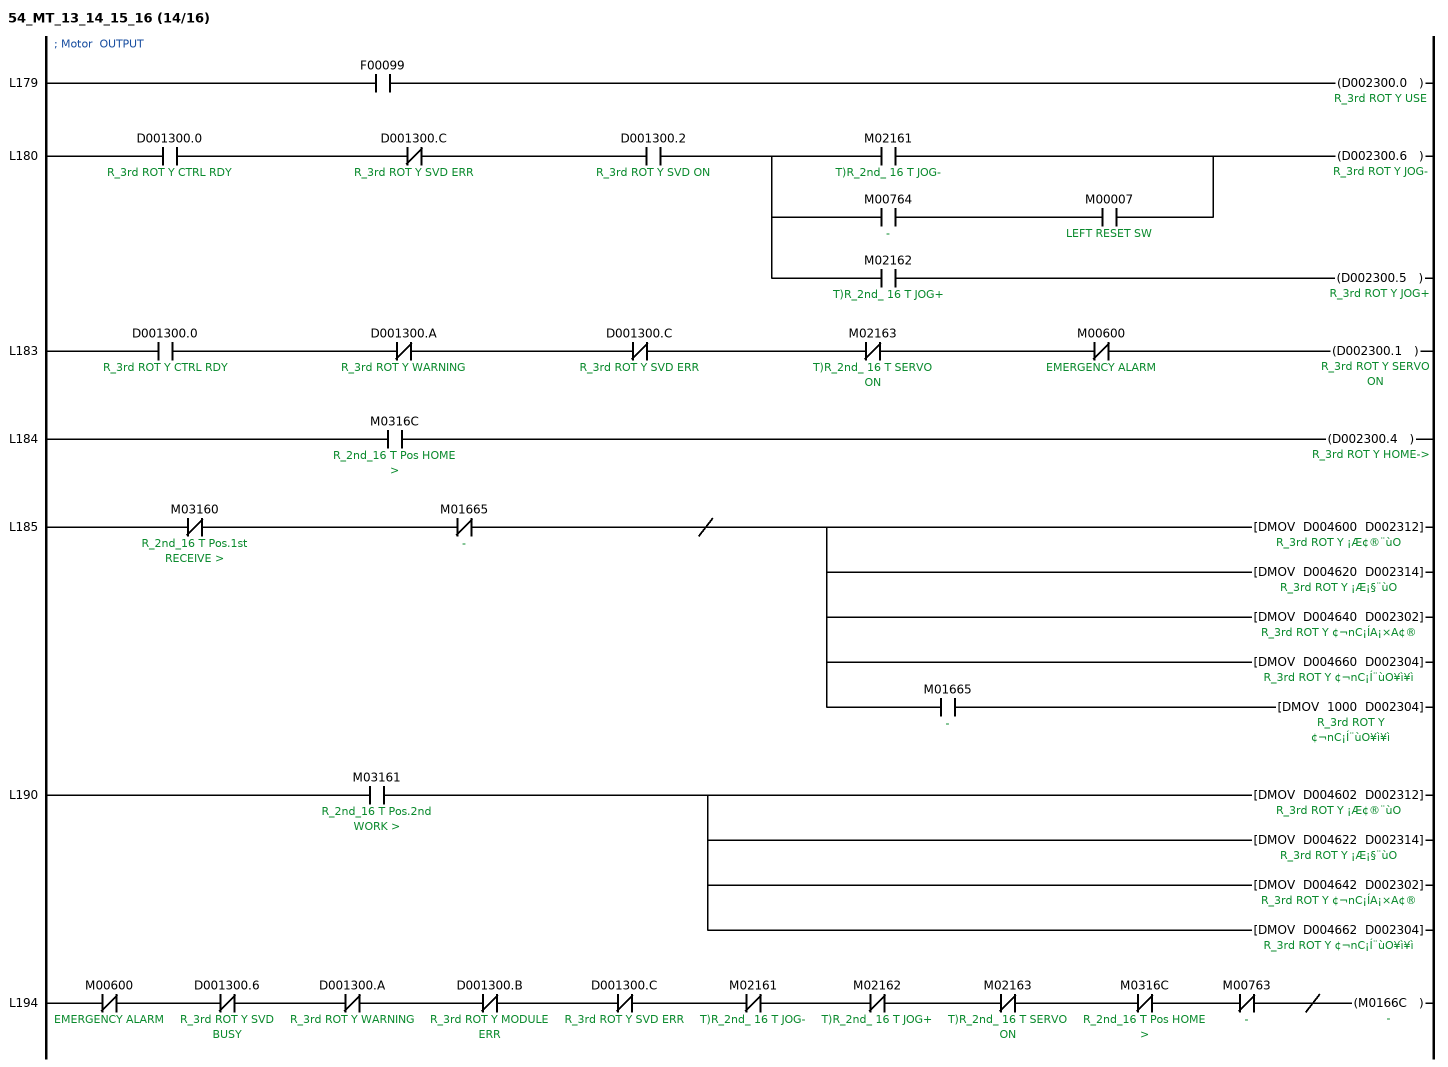
[picture p312: 54_MT_13_14_15_16 rungs L179-L194]
//  Motor  OUTPUT
; L179
LOAD      F00099
OUT       D002300.0	// R_3rd ROT Y USE
; L180
LOAD      D001300.0	// R_3rd ROT Y CTRL RDY
AND NOT   D001300.C	// R_3rd ROT Y SVD ERR
AND       D001300.2	// R_3rd ROT Y SVD ON
MPUSH
LOAD      M02161	// T)R_2nd_ 16 T JOG-
LOAD      M00764	// -
AND       M00007	// LEFT RESET SW
OR LOAD
AND LOAD
OUT       D002300.6	// R_3rd ROT Y JOG-
MPOP
AND       M02162	// T)R_2nd_ 16 T JOG+
OUT       D002300.5	// R_3rd ROT Y JOG+
; L183
LOAD      D001300.0	// R_3rd ROT Y CTRL RDY
AND NOT   D001300.A	// R_3rd ROT Y WARNING
AND NOT   D001300.C	// R_3rd ROT Y SVD ERR
AND NOT   M02163	// T)R_2nd_ 16 T SERVO ON
AND NOT   M00600	// EMERGENCY ALARM
OUT       D002300.1	// R_3rd ROT Y SERVO ON
; L184
LOAD      M0316C	// R_2nd_16 T Pos HOME >
OUT       D002300.4	// R_3rd ROT Y HOME->
; L185
LOAD NOT  M03160	// R_2nd_16 T Pos.1st RECEIVE >
AND NOT   M01665	// -
NOT
DMOV      D004600 D002312	// R_3rd ROT Y ¡Æ¢®¨ùO
DMOV      D004620 D002314	// R_3rd ROT Y ¡Æ¡§¨ùO
DMOV      D004640 D002302	// R_3rd ROT Y ¢¬nC¡ÍA¡×A¢®
DMOV      D004660 D002304	// R_3rd ROT Y ¢¬nC¡Í¨ùO¥ì¥ì
AND       M01665	// -
DMOV      1000 D002304	// R_3rd ROT Y ¢¬nC¡Í¨ùO¥ì¥ì
; L190
LOAD      M03161	// R_2nd_16 T Pos.2nd WORK >
DMOV      D004602 D002312	// R_3rd ROT Y ¡Æ¢®¨ùO
DMOV      D004622 D002314	// R_3rd ROT Y ¡Æ¡§¨ùO
DMOV      D004642 D002302	// R_3rd ROT Y ¢¬nC¡ÍA¡×A¢®
DMOV      D004662 D002304	// R_3rd ROT Y ¢¬nC¡Í¨ùO¥ì¥ì
; L194
LOAD NOT  M00600	// EMERGENCY ALARM
AND NOT   D001300.6	// R_3rd ROT Y SVD BUSY
AND NOT   D001300.A	// R_3rd ROT Y WARNING
AND NOT   D001300.B	// R_3rd ROT Y MODULE ERR
AND NOT   D001300.C	// R_3rd ROT Y SVD ERR
AND NOT   M02161	// T)R_2nd_ 16 T JOG-
AND NOT   M02162	// T)R_2nd_ 16 T JOG+
AND NOT   M02163	// T)R_2nd_ 16 T SERVO ON
AND NOT   M0316C	// R_2nd_16 T Pos HOME >
AND NOT   M00763	// -
NOT
OUT       M0166C	// -

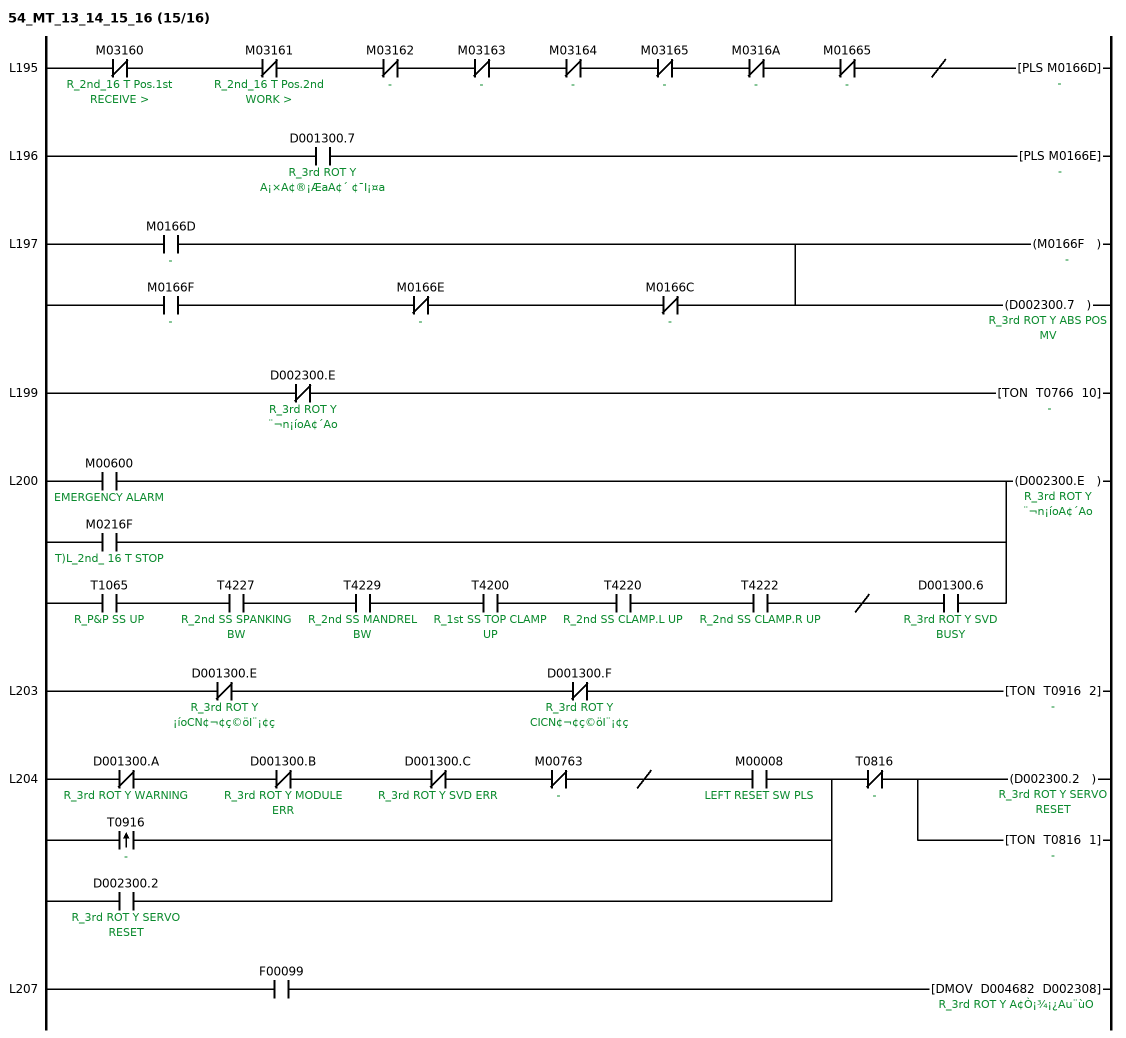
; L195
LOAD NOT  M03160	// R_2nd_16 T Pos.1st RECEIVE >
AND NOT   M03161	// R_2nd_16 T Pos.2nd WORK >
AND NOT   M03162	// -
AND NOT   M03163	// -
AND NOT   M03164	// -
AND NOT   M03165	// -
AND NOT   M0316A	// -
AND NOT   M01665	// -
NOT
OUTP      M0166D	// -
; L196
LOAD      D001300.7	// R_3rd ROT Y A¡×A¢®¡ÆaA¢´ ¢¯I¡¤a
OUTP      M0166E	// -
; L197
LOAD      M0166D	// -
LOAD      M0166F	// -
AND NOT   M0166E	// -
AND NOT   M0166C	// -
OR LOAD
OUT       M0166F	// -
OUT       D002300.7	// R_3rd ROT Y ABS POS MV
; L199
LOAD NOT  D002300.E	// R_3rd ROT Y ¨¬n¡íoA¢´Ao
TON       T0766 10	// -
; L200
LOAD      M00600	// EMERGENCY ALARM
OR        M0216F	// T)L_2nd_ 16 T STOP
LOAD      T1065	// R_P&P SS UP
AND       T4227	// R_2nd SS SPANKING BW
AND       T4229	// R_2nd SS MANDREL BW
AND       T4200	// R_1st SS TOP CLAMP UP
AND       T4220	// R_2nd SS CLAMP.L UP
AND       T4222	// R_2nd SS CLAMP.R UP
NOT
AND       D001300.6	// R_3rd ROT Y SVD BUSY
OR LOAD
OUT       D002300.E	// R_3rd ROT Y ¨¬n¡íoA¢´Ao
; L203
LOAD NOT  D001300.E	// R_3rd ROT Y ¡íoCN¢¬¢ç©öI¨¡¢ç
AND NOT   D001300.F	// R_3rd ROT Y CICN¢¬¢ç©öI¨¡¢ç
TON       T0916 2	// -
; L204
LOAD NOT  D001300.A	// R_3rd ROT Y WARNING
AND NOT   D001300.B	// R_3rd ROT Y MODULE ERR
AND NOT   D001300.C	// R_3rd ROT Y SVD ERR
AND NOT   M00763	// -
NOT
AND       M00008	// LEFT RESET SW PLS
ORP       T0916	// -
OR        D002300.2	// R_3rd ROT Y SERVO RESET
AND NOT   T0816	// -
OUT       D002300.2	// R_3rd ROT Y SERVO RESET
TON       T0816 1	// -
; L207
LOAD      F00099
DMOV      D004682 D002308	// R_3rd ROT Y A¢Ò¡¾¡¿Au¨ùO

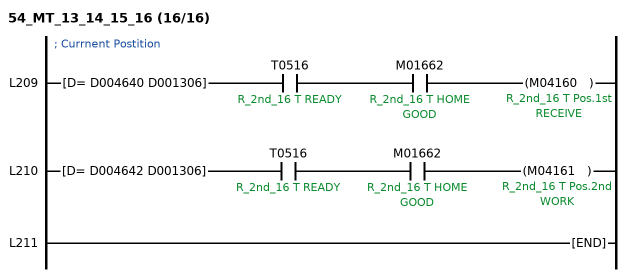
// Currnent Postition
; L209
LOADD=    D004640 D001306
AND       T0516	// R_2nd_16 T READY
AND       M01662	// R_2nd_16 T HOME GOOD
OUT       M04160	// R_2nd_16 T Pos.1st RECEIVE
; L210
LOADD=    D004642 D001306
AND       T0516	// R_2nd_16 T READY
AND       M01662	// R_2nd_16 T HOME GOOD
OUT       M04161	// R_2nd_16 T Pos.2nd WORK
; L211
END

PROGRAM 55_MT_17_18_19_20 (task: ¨ö¨¬A¥ì CA¡¤I¡¾¡¿¡¤¡Í)

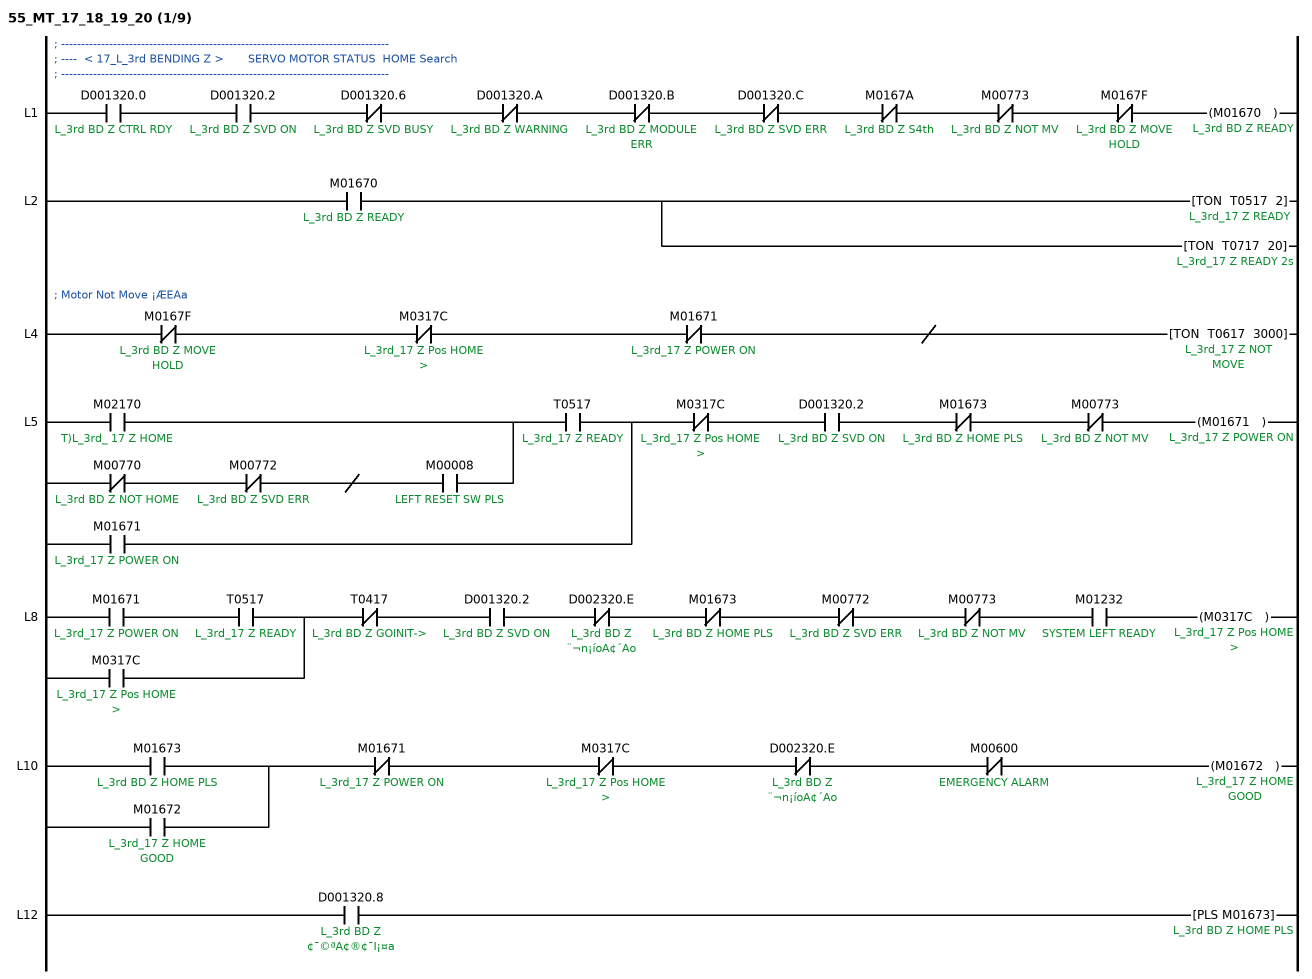
// ----------------------------------------------------------------------------------
// 
// ----  < 17_L_3rd BENDING Z >       SERVO MOTOR STATUS  HOME Search
// 
// ----------------------------------------------------------------------------------
; L1
LOAD      D001320.0	// L_3rd BD Z CTRL RDY
AND       D001320.2	// L_3rd BD Z SVD ON
AND NOT   D001320.6	// L_3rd BD Z SVD BUSY
AND NOT   D001320.A	// L_3rd BD Z WARNING
AND NOT   D001320.B	// L_3rd BD Z MODULE ERR
AND NOT   D001320.C	// L_3rd BD Z SVD ERR
AND NOT   M0167A	// L_3rd BD Z S4th
AND NOT   M00773	// L_3rd BD Z NOT MV
AND NOT   M0167F	// L_3rd BD Z MOVE HOLD
OUT       M01670	// L_3rd BD Z READY
; L2
LOAD      M01670	// L_3rd BD Z READY
TON       T0517 2	// L_3rd_17 Z READY
TON       T0717 20	// L_3rd_17 Z READY 2s
; L4
LOAD NOT  M0167F	// L_3rd BD Z MOVE HOLD
AND NOT   M0317C	// L_3rd_17 Z Pos HOME >
AND NOT   M01671	// L_3rd_17 Z POWER ON
NOT
TON       T0617 3000	// L_3rd_17 Z NOT MOVE
// output comment: Motor Not Move ¡ÆEAa
; L5
LOAD      M02170	// T)L_3rd_ 17 Z HOME
LOAD NOT  M00770	// L_3rd BD Z NOT HOME
AND NOT   M00772	// L_3rd BD Z SVD ERR
NOT
AND       M00008	// LEFT RESET SW PLS
OR LOAD
AND       T0517	// L_3rd_17 Z READY
OR        M01671	// L_3rd_17 Z POWER ON
AND NOT   M0317C	// L_3rd_17 Z Pos HOME >
AND       D001320.2	// L_3rd BD Z SVD ON
AND NOT   M01673	// L_3rd BD Z HOME PLS
AND NOT   M00773	// L_3rd BD Z NOT MV
OUT       M01671	// L_3rd_17 Z POWER ON
; L8
LOAD      M01671	// L_3rd_17 Z POWER ON
AND       T0517	// L_3rd_17 Z READY
OR        M0317C	// L_3rd_17 Z Pos HOME >
AND NOT   T0417	// L_3rd BD Z GOINIT->
AND       D001320.2	// L_3rd BD Z SVD ON
AND NOT   D002320.E	// L_3rd BD Z ¨¬n¡íoA¢´Ao
AND NOT   M01673	// L_3rd BD Z HOME PLS
AND NOT   M00772	// L_3rd BD Z SVD ERR
AND NOT   M00773	// L_3rd BD Z NOT MV
AND       M01232	// SYSTEM LEFT READY
OUT       M0317C	// L_3rd_17 Z Pos HOME >
; L10
LOAD      M01673	// L_3rd BD Z HOME PLS
OR        M01672	// L_3rd_17 Z HOME GOOD
AND NOT   M01671	// L_3rd_17 Z POWER ON
AND NOT   M0317C	// L_3rd_17 Z Pos HOME >
AND NOT   D002320.E	// L_3rd BD Z ¨¬n¡íoA¢´Ao
AND NOT   M00600	// EMERGENCY ALARM
OUT       M01672	// L_3rd_17 Z HOME GOOD
; L12
LOAD      D001320.8	// L_3rd BD Z ¢¯©ªA¢®¢¯I¡¤a
OUTP      M01673	// L_3rd BD Z HOME PLS

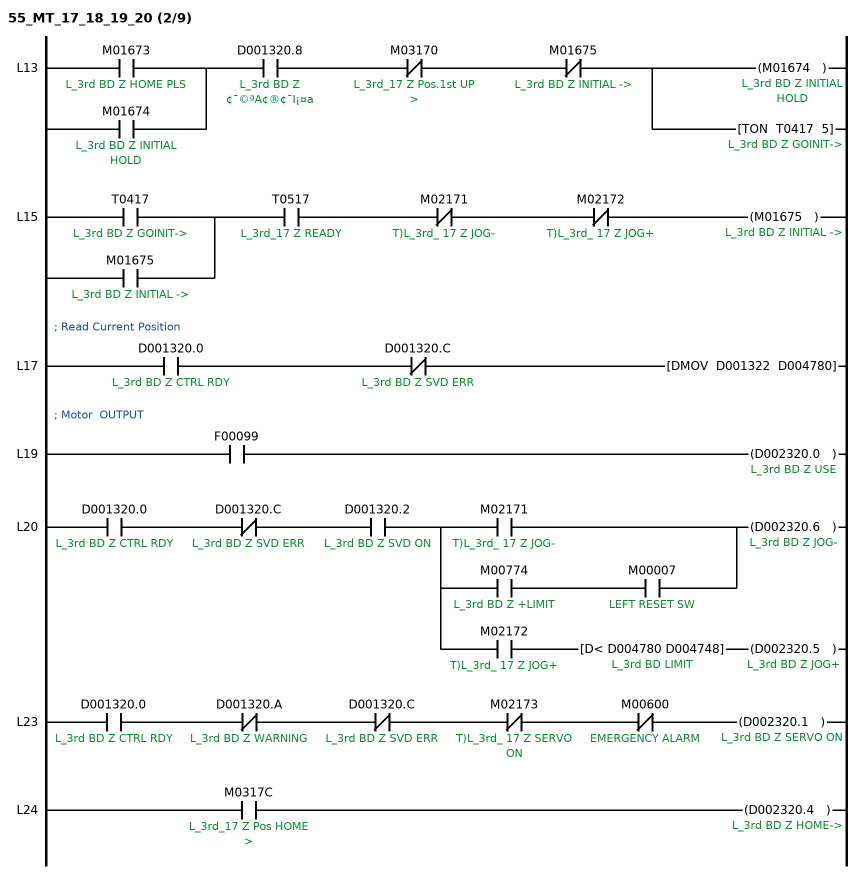
; L13
LOAD      M01673	// L_3rd BD Z HOME PLS
OR        M01674	// L_3rd BD Z INITIAL HOLD
AND       D001320.8	// L_3rd BD Z ¢¯©ªA¢®¢¯I¡¤a
AND NOT   M03170	// L_3rd_17 Z Pos.1st UP >
AND NOT   M01675	// L_3rd BD Z INITIAL ->
OUT       M01674	// L_3rd BD Z INITIAL HOLD
TON       T0417 5	// L_3rd BD Z GOINIT->
; L15
LOAD      T0417	// L_3rd BD Z GOINIT->
OR        M01675	// L_3rd BD Z INITIAL ->
AND       T0517	// L_3rd_17 Z READY
AND NOT   M02171	// T)L_3rd_ 17 Z JOG-
AND NOT   M02172	// T)L_3rd_ 17 Z JOG+
OUT       M01675	// L_3rd BD Z INITIAL ->
; L17
LOAD      D001320.0	// L_3rd BD Z CTRL RDY
AND NOT   D001320.C	// L_3rd BD Z SVD ERR
DMOV      D001322 D004780
// output comment: Read Current Position
//  Motor  OUTPUT
; L19
LOAD      F00099
OUT       D002320.0	// L_3rd BD Z USE
; L20
LOAD      D001320.0	// L_3rd BD Z CTRL RDY
AND NOT   D001320.C	// L_3rd BD Z SVD ERR
AND       D001320.2	// L_3rd BD Z SVD ON
MPUSH
LOAD      M02171	// T)L_3rd_ 17 Z JOG-
LOAD      M00774	// L_3rd BD Z +LIMIT
AND       M00007	// LEFT RESET SW
OR LOAD
AND LOAD
OUT       D002320.6	// L_3rd BD Z JOG-
MPOP
AND       M02172	// T)L_3rd_ 17 Z JOG+
ANDD<     D004780 D004748	// L_3rd BD LIMIT
OUT       D002320.5	// L_3rd BD Z JOG+
; L23
LOAD      D001320.0	// L_3rd BD Z CTRL RDY
AND NOT   D001320.A	// L_3rd BD Z WARNING
AND NOT   D001320.C	// L_3rd BD Z SVD ERR
AND NOT   M02173	// T)L_3rd_ 17 Z SERVO ON
AND NOT   M00600	// EMERGENCY ALARM
OUT       D002320.1	// L_3rd BD Z SERVO ON
; L24
LOAD      M0317C	// L_3rd_17 Z Pos HOME >
OUT       D002320.4	// L_3rd BD Z HOME->

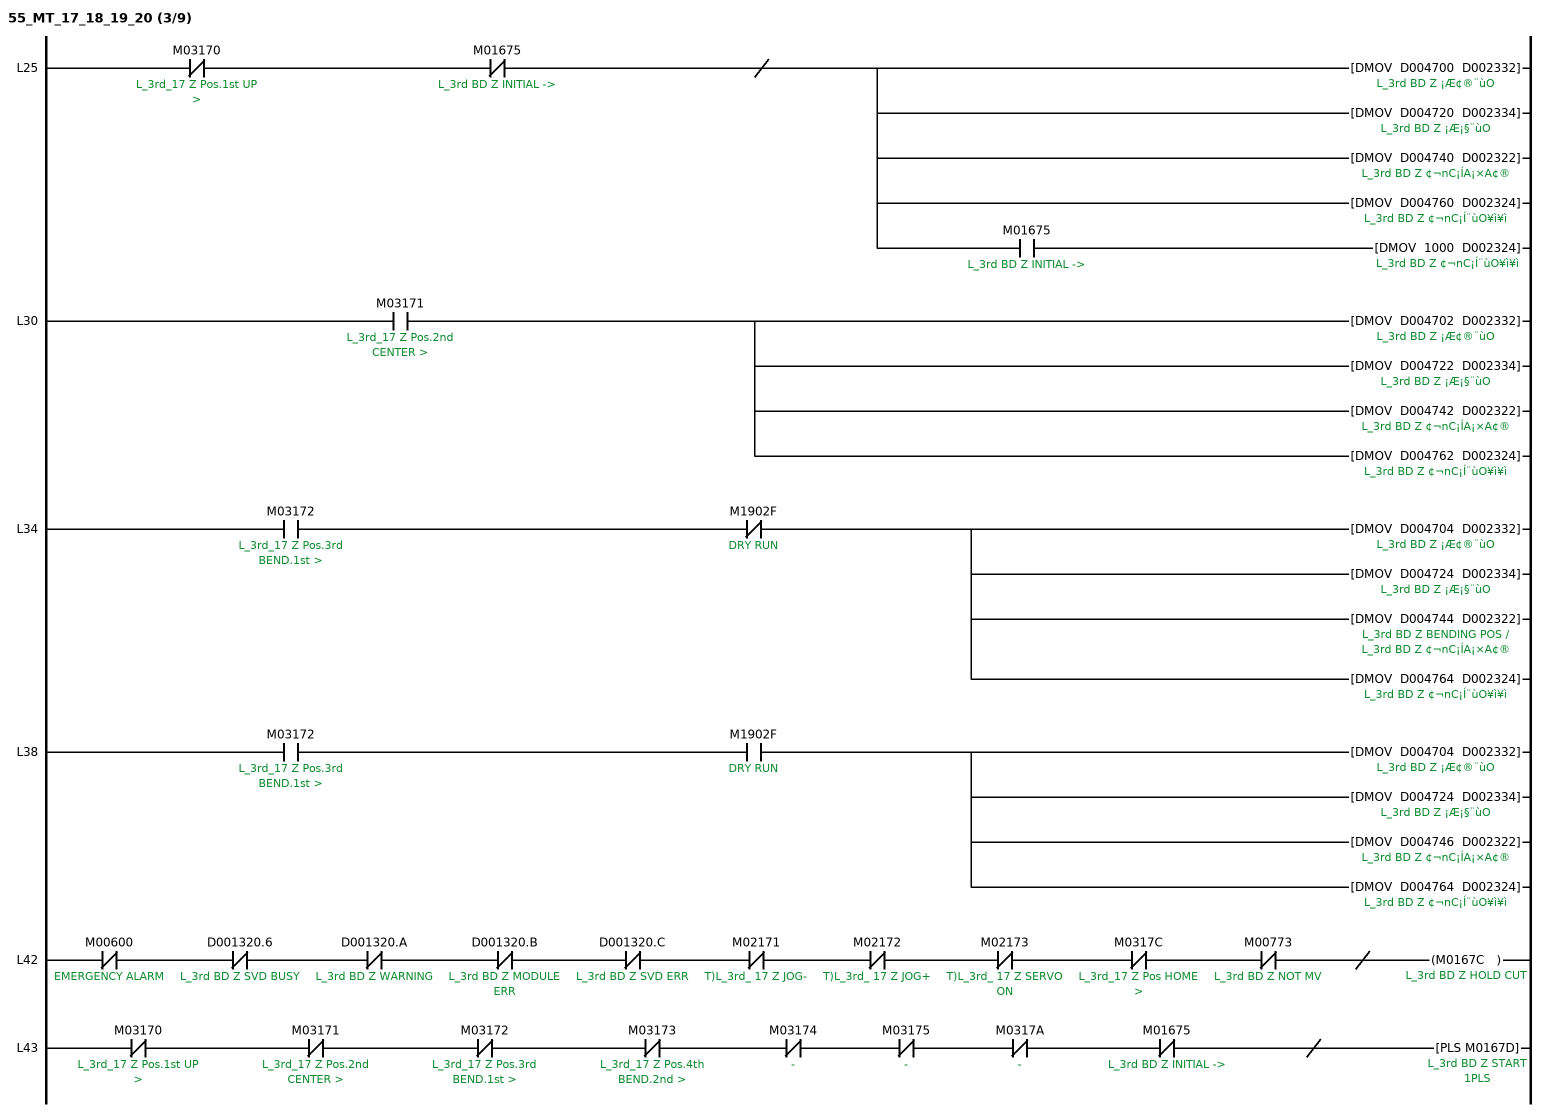
; L25
LOAD NOT  M03170	// L_3rd_17 Z Pos.1st UP >
AND NOT   M01675	// L_3rd BD Z INITIAL ->
NOT
DMOV      D004700 D002332	// L_3rd BD Z ¡Æ¢®¨ùO
DMOV      D004720 D002334	// L_3rd BD Z ¡Æ¡§¨ùO
DMOV      D004740 D002322	// L_3rd BD Z ¢¬nC¡ÍA¡×A¢®
DMOV      D004760 D002324	// L_3rd BD Z ¢¬nC¡Í¨ùO¥ì¥ì
AND       M01675	// L_3rd BD Z INITIAL ->
DMOV      1000 D002324	// L_3rd BD Z ¢¬nC¡Í¨ùO¥ì¥ì
; L30
LOAD      M03171	// L_3rd_17 Z Pos.2nd CENTER >
DMOV      D004702 D002332	// L_3rd BD Z ¡Æ¢®¨ùO
DMOV      D004722 D002334	// L_3rd BD Z ¡Æ¡§¨ùO
DMOV      D004742 D002322	// L_3rd BD Z ¢¬nC¡ÍA¡×A¢®
DMOV      D004762 D002324	// L_3rd BD Z ¢¬nC¡Í¨ùO¥ì¥ì
; L34
LOAD      M03172	// L_3rd_17 Z Pos.3rd BEND.1st >
AND NOT   M1902F	// DRY RUN
DMOV      D004704 D002332	// L_3rd BD Z ¡Æ¢®¨ùO
DMOV      D004724 D002334	// L_3rd BD Z ¡Æ¡§¨ùO
DMOV      D004744 D002322	// L_3rd BD Z BENDING POS / L_3rd BD Z ¢¬nC¡ÍA¡×A¢®
DMOV      D004764 D002324	// L_3rd BD Z ¢¬nC¡Í¨ùO¥ì¥ì
; L38
LOAD      M03172	// L_3rd_17 Z Pos.3rd BEND.1st >
AND       M1902F	// DRY RUN
DMOV      D004704 D002332	// L_3rd BD Z ¡Æ¢®¨ùO
DMOV      D004724 D002334	// L_3rd BD Z ¡Æ¡§¨ùO
DMOV      D004746 D002322	// L_3rd BD Z ¢¬nC¡ÍA¡×A¢®
DMOV      D004764 D002324	// L_3rd BD Z ¢¬nC¡Í¨ùO¥ì¥ì
; L42
LOAD NOT  M00600	// EMERGENCY ALARM
AND NOT   D001320.6	// L_3rd BD Z SVD BUSY
AND NOT   D001320.A	// L_3rd BD Z WARNING
AND NOT   D001320.B	// L_3rd BD Z MODULE ERR
AND NOT   D001320.C	// L_3rd BD Z SVD ERR
AND NOT   M02171	// T)L_3rd_ 17 Z JOG-
AND NOT   M02172	// T)L_3rd_ 17 Z JOG+
AND NOT   M02173	// T)L_3rd_ 17 Z SERVO ON
AND NOT   M0317C	// L_3rd_17 Z Pos HOME >
AND NOT   M00773	// L_3rd BD Z NOT MV
NOT
OUT       M0167C	// L_3rd BD Z HOLD CUT
; L43
LOAD NOT  M03170	// L_3rd_17 Z Pos.1st UP >
AND NOT   M03171	// L_3rd_17 Z Pos.2nd CENTER >
AND NOT   M03172	// L_3rd_17 Z Pos.3rd BEND.1st >
AND NOT   M03173	// L_3rd_17 Z Pos.4th BEND.2nd >
AND NOT   M03174	// -
AND NOT   M03175	// -
AND NOT   M0317A	// -
AND NOT   M01675	// L_3rd BD Z INITIAL ->
NOT
OUTP      M0167D	// L_3rd BD Z START 1PLS

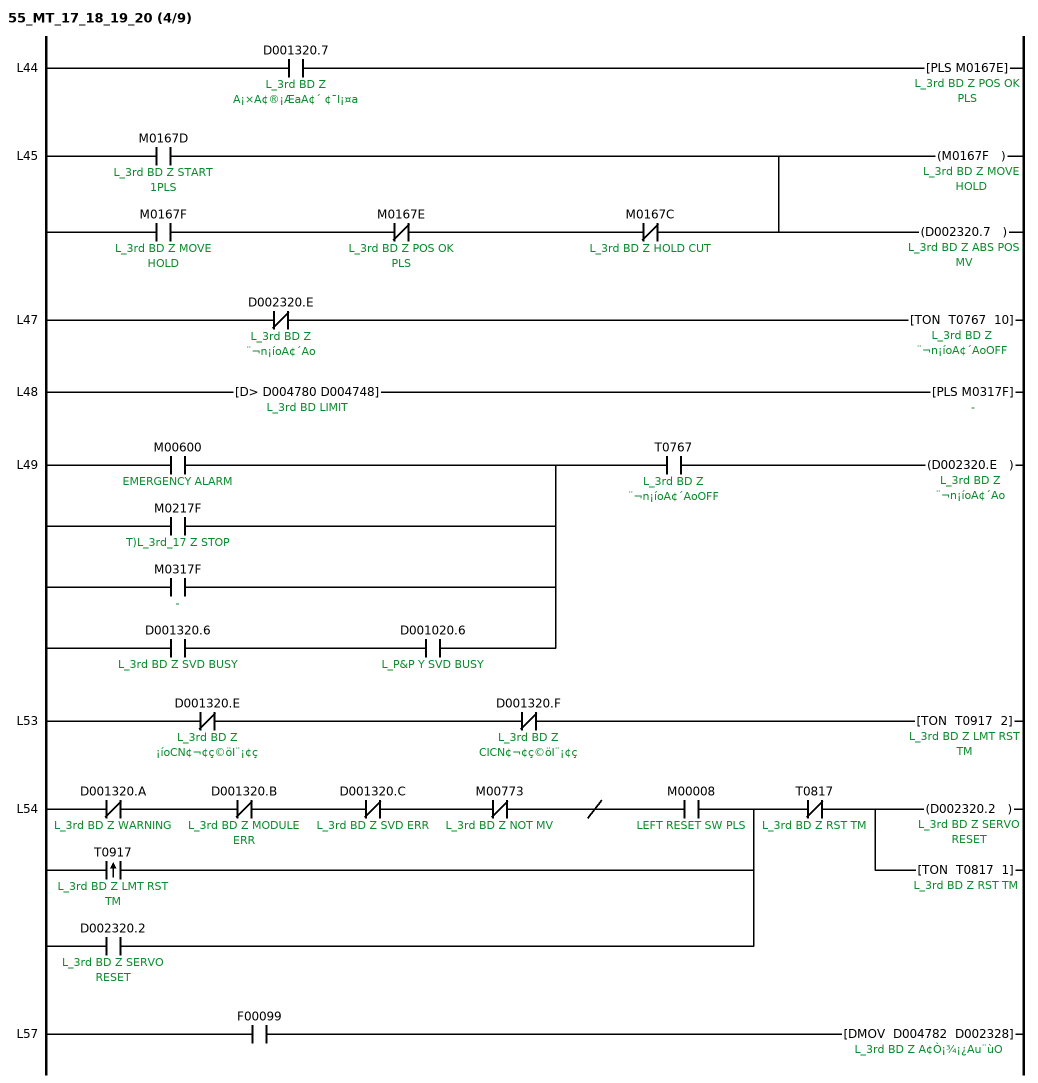
; L44
LOAD      D001320.7	// L_3rd BD Z A¡×A¢®¡ÆaA¢´ ¢¯I¡¤a
OUTP      M0167E	// L_3rd BD Z POS OK PLS
; L45
LOAD      M0167D	// L_3rd BD Z START 1PLS
LOAD      M0167F	// L_3rd BD Z MOVE HOLD
AND NOT   M0167E	// L_3rd BD Z POS OK PLS
AND NOT   M0167C	// L_3rd BD Z HOLD CUT
OR LOAD
OUT       M0167F	// L_3rd BD Z MOVE HOLD
OUT       D002320.7	// L_3rd BD Z ABS POS MV
; L47
LOAD NOT  D002320.E	// L_3rd BD Z ¨¬n¡íoA¢´Ao
TON       T0767 10	// L_3rd BD Z ¨¬n¡íoA¢´AoOFF
; L48
LOADD>    D004780 D004748	// L_3rd BD LIMIT
OUTP      M0317F	// -
; L49
LOAD      M00600	// EMERGENCY ALARM
OR        M0217F	// T)L_3rd_17 Z STOP
OR        M0317F	// -
LOAD      D001320.6	// L_3rd BD Z SVD BUSY
AND       D001020.6	// L_P&P Y SVD BUSY
OR LOAD
AND       T0767	// L_3rd BD Z ¨¬n¡íoA¢´AoOFF
OUT       D002320.E	// L_3rd BD Z ¨¬n¡íoA¢´Ao
; L53
LOAD NOT  D001320.E	// L_3rd BD Z ¡íoCN¢¬¢ç©öI¨¡¢ç
AND NOT   D001320.F	// L_3rd BD Z CICN¢¬¢ç©öI¨¡¢ç
TON       T0917 2	// L_3rd BD Z LMT RST TM
; L54
LOAD NOT  D001320.A	// L_3rd BD Z WARNING
AND NOT   D001320.B	// L_3rd BD Z MODULE ERR
AND NOT   D001320.C	// L_3rd BD Z SVD ERR
AND NOT   M00773	// L_3rd BD Z NOT MV
NOT
AND       M00008	// LEFT RESET SW PLS
ORP       T0917	// L_3rd BD Z LMT RST TM
OR        D002320.2	// L_3rd BD Z SERVO RESET
AND NOT   T0817	// L_3rd BD Z RST TM
OUT       D002320.2	// L_3rd BD Z SERVO RESET
TON       T0817 1	// L_3rd BD Z RST TM
; L57
LOAD      F00099
DMOV      D004782 D002328	// L_3rd BD Z A¢Ò¡¾¡¿Au¨ùO

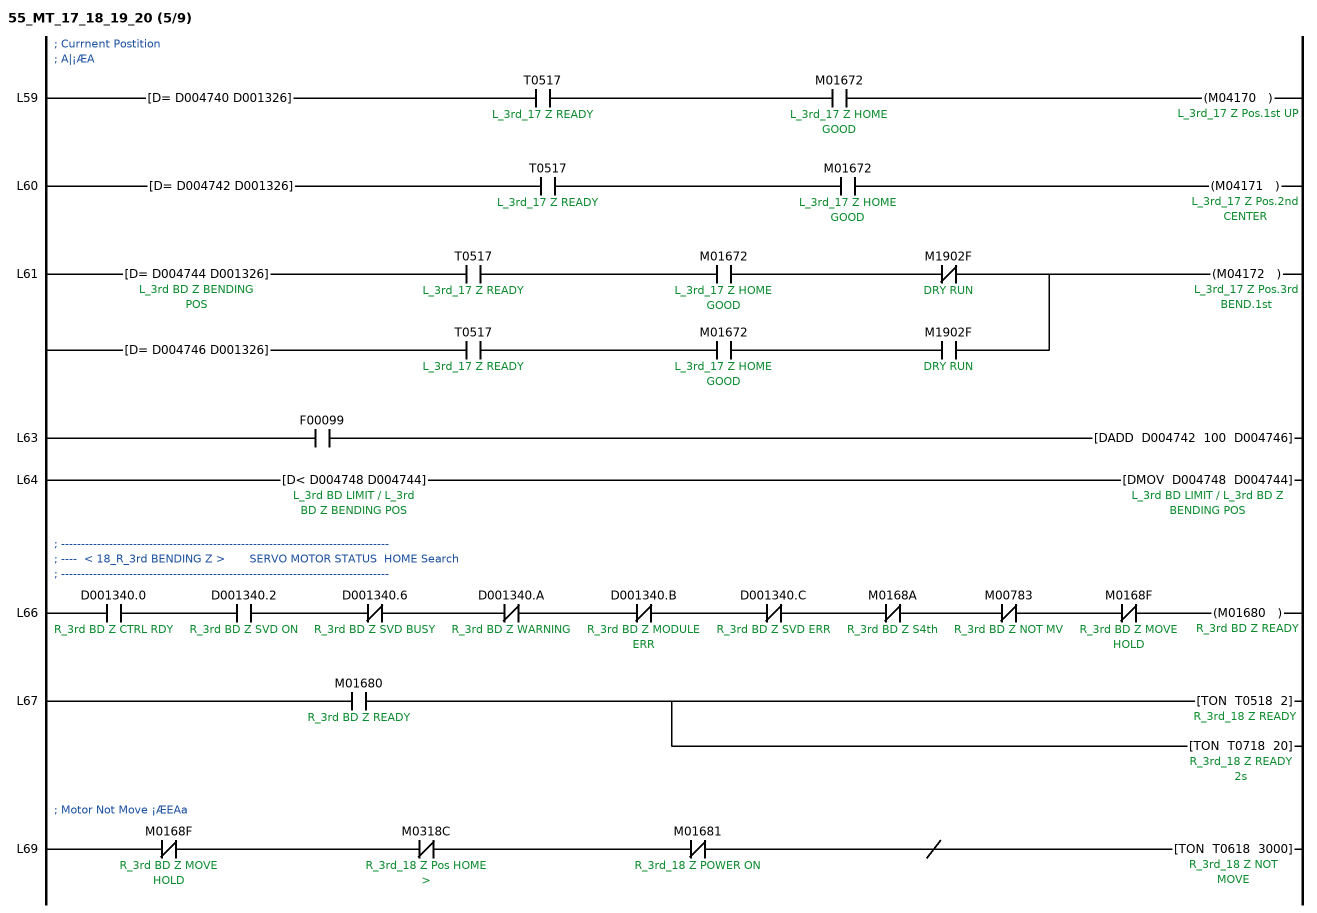
// Currnent Postition
; L59
LOADD=    D004740 D001326
AND       T0517	// L_3rd_17 Z READY
AND       M01672	// L_3rd_17 Z HOME GOOD
OUT       M04170	// L_3rd_17 Z Pos.1st UP
// output comment: A|¡ÆA
; L60
LOADD=    D004742 D001326
AND       T0517	// L_3rd_17 Z READY
AND       M01672	// L_3rd_17 Z HOME GOOD
OUT       M04171	// L_3rd_17 Z Pos.2nd CENTER
; L61
LOADD=    D004744 D001326	// L_3rd BD Z BENDING POS
AND       T0517	// L_3rd_17 Z READY
AND       M01672	// L_3rd_17 Z HOME GOOD
AND NOT   M1902F	// DRY RUN
LOADD=    D004746 D001326
AND       T0517	// L_3rd_17 Z READY
AND       M01672	// L_3rd_17 Z HOME GOOD
AND       M1902F	// DRY RUN
OR LOAD
OUT       M04172	// L_3rd_17 Z Pos.3rd BEND.1st
; L63
LOAD      F00099
DADD      D004742 100 D004746
; L64
LOADD<    D004748 D004744	// L_3rd BD LIMIT / L_3rd BD Z BENDING POS
DMOV      D004748 D004744	// L_3rd BD LIMIT / L_3rd BD Z BENDING POS
// ----------------------------------------------------------------------------------
// 
// ----  < 18_R_3rd BENDING Z >       SERVO MOTOR STATUS  HOME Search
// 
// ----------------------------------------------------------------------------------
; L66
LOAD      D001340.0	// R_3rd BD Z CTRL RDY
AND       D001340.2	// R_3rd BD Z SVD ON
AND NOT   D001340.6	// R_3rd BD Z SVD BUSY
AND NOT   D001340.A	// R_3rd BD Z WARNING
AND NOT   D001340.B	// R_3rd BD Z MODULE ERR
AND NOT   D001340.C	// R_3rd BD Z SVD ERR
AND NOT   M0168A	// R_3rd BD Z S4th
AND NOT   M00783	// R_3rd BD Z NOT MV
AND NOT   M0168F	// R_3rd BD Z MOVE HOLD
OUT       M01680	// R_3rd BD Z READY
; L67
LOAD      M01680	// R_3rd BD Z READY
TON       T0518 2	// R_3rd_18 Z READY
TON       T0718 20	// R_3rd_18 Z READY 2s
; L69
LOAD NOT  M0168F	// R_3rd BD Z MOVE HOLD
AND NOT   M0318C	// R_3rd_18 Z Pos HOME >
AND NOT   M01681	// R_3rd_18 Z POWER ON
NOT
TON       T0618 3000	// R_3rd_18 Z NOT MOVE
// output comment: Motor Not Move ¡ÆEAa

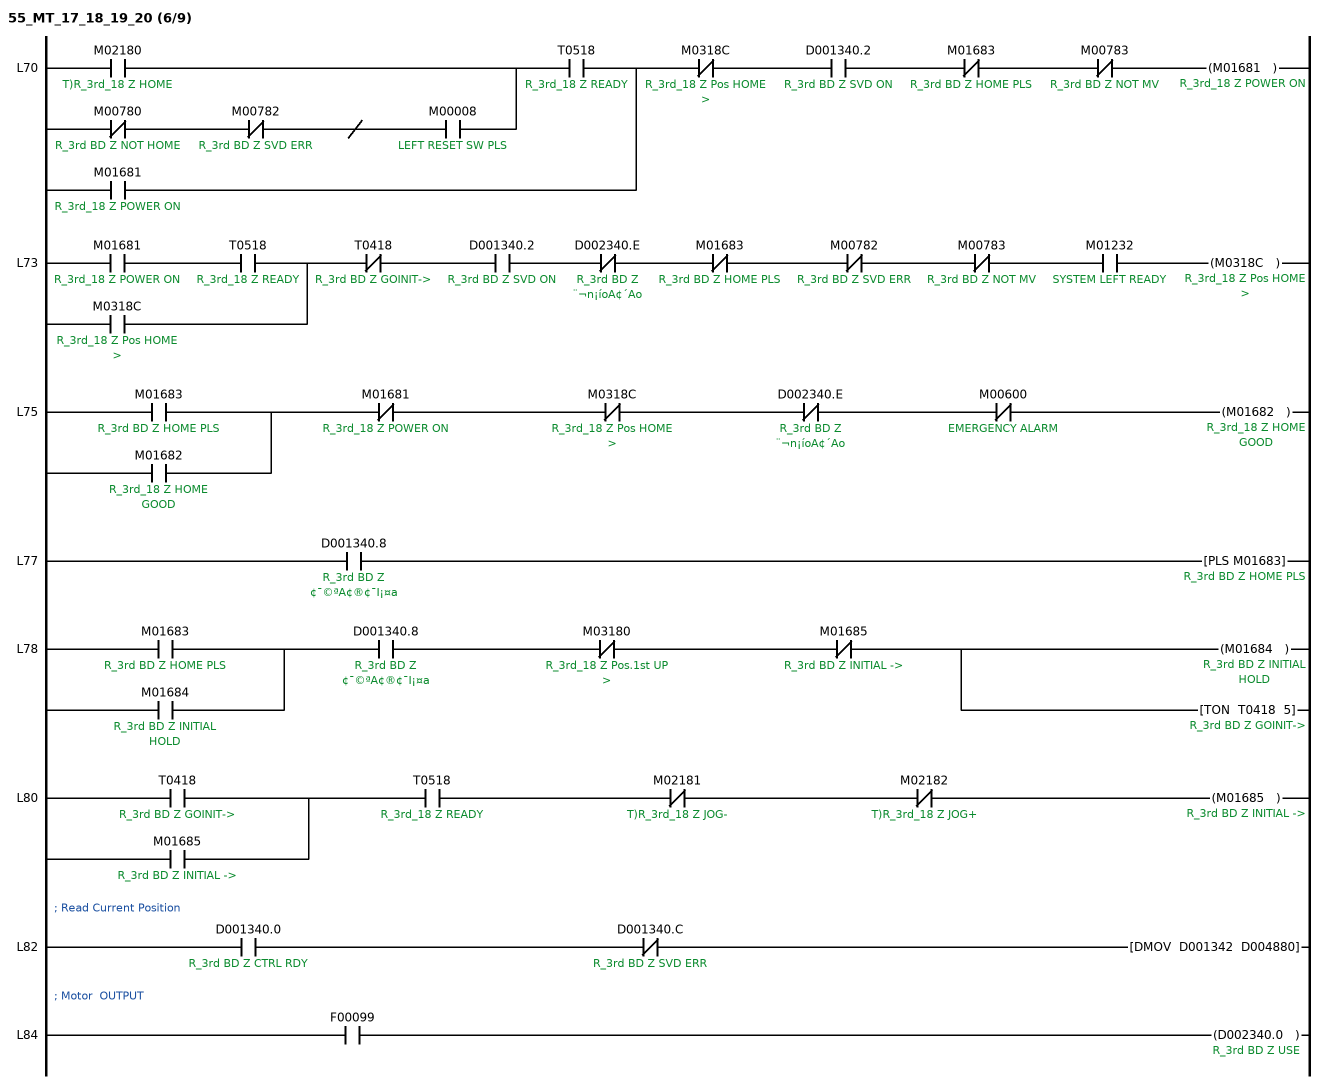
; L70
LOAD      M02180	// T)R_3rd_18 Z HOME
LOAD NOT  M00780	// R_3rd BD Z NOT HOME
AND NOT   M00782	// R_3rd BD Z SVD ERR
NOT
AND       M00008	// LEFT RESET SW PLS
OR LOAD
AND       T0518	// R_3rd_18 Z READY
OR        M01681	// R_3rd_18 Z POWER ON
AND NOT   M0318C	// R_3rd_18 Z Pos HOME >
AND       D001340.2	// R_3rd BD Z SVD ON
AND NOT   M01683	// R_3rd BD Z HOME PLS
AND NOT   M00783	// R_3rd BD Z NOT MV
OUT       M01681	// R_3rd_18 Z POWER ON
; L73
LOAD      M01681	// R_3rd_18 Z POWER ON
AND       T0518	// R_3rd_18 Z READY
OR        M0318C	// R_3rd_18 Z Pos HOME >
AND NOT   T0418	// R_3rd BD Z GOINIT->
AND       D001340.2	// R_3rd BD Z SVD ON
AND NOT   D002340.E	// R_3rd BD Z ¨¬n¡íoA¢´Ao
AND NOT   M01683	// R_3rd BD Z HOME PLS
AND NOT   M00782	// R_3rd BD Z SVD ERR
AND NOT   M00783	// R_3rd BD Z NOT MV
AND       M01232	// SYSTEM LEFT READY
OUT       M0318C	// R_3rd_18 Z Pos HOME >
; L75
LOAD      M01683	// R_3rd BD Z HOME PLS
OR        M01682	// R_3rd_18 Z HOME GOOD
AND NOT   M01681	// R_3rd_18 Z POWER ON
AND NOT   M0318C	// R_3rd_18 Z Pos HOME >
AND NOT   D002340.E	// R_3rd BD Z ¨¬n¡íoA¢´Ao
AND NOT   M00600	// EMERGENCY ALARM
OUT       M01682	// R_3rd_18 Z HOME GOOD
; L77
LOAD      D001340.8	// R_3rd BD Z ¢¯©ªA¢®¢¯I¡¤a
OUTP      M01683	// R_3rd BD Z HOME PLS
; L78
LOAD      M01683	// R_3rd BD Z HOME PLS
OR        M01684	// R_3rd BD Z INITIAL HOLD
AND       D001340.8	// R_3rd BD Z ¢¯©ªA¢®¢¯I¡¤a
AND NOT   M03180	// R_3rd_18 Z Pos.1st UP >
AND NOT   M01685	// R_3rd BD Z INITIAL ->
OUT       M01684	// R_3rd BD Z INITIAL HOLD
TON       T0418 5	// R_3rd BD Z GOINIT->
; L80
LOAD      T0418	// R_3rd BD Z GOINIT->
OR        M01685	// R_3rd BD Z INITIAL ->
AND       T0518	// R_3rd_18 Z READY
AND NOT   M02181	// T)R_3rd_18 Z JOG-
AND NOT   M02182	// T)R_3rd_18 Z JOG+
OUT       M01685	// R_3rd BD Z INITIAL ->
; L82
LOAD      D001340.0	// R_3rd BD Z CTRL RDY
AND NOT   D001340.C	// R_3rd BD Z SVD ERR
DMOV      D001342 D004880
// output comment: Read Current Position
//  Motor  OUTPUT
; L84
LOAD      F00099
OUT       D002340.0	// R_3rd BD Z USE

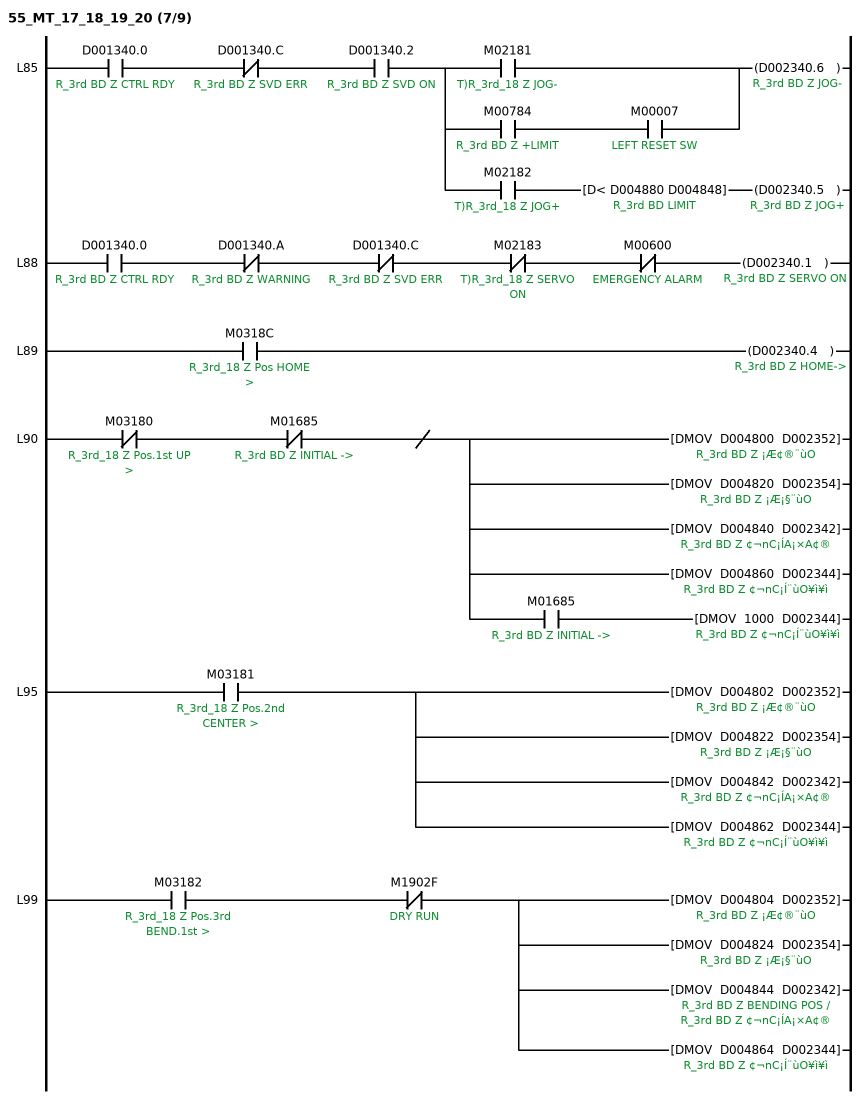
; L85
LOAD      D001340.0	// R_3rd BD Z CTRL RDY
AND NOT   D001340.C	// R_3rd BD Z SVD ERR
AND       D001340.2	// R_3rd BD Z SVD ON
MPUSH
LOAD      M02181	// T)R_3rd_18 Z JOG-
LOAD      M00784	// R_3rd BD Z +LIMIT
AND       M00007	// LEFT RESET SW
OR LOAD
AND LOAD
OUT       D002340.6	// R_3rd BD Z JOG-
MPOP
AND       M02182	// T)R_3rd_18 Z JOG+
ANDD<     D004880 D004848	// R_3rd BD LIMIT
OUT       D002340.5	// R_3rd BD Z JOG+
; L88
LOAD      D001340.0	// R_3rd BD Z CTRL RDY
AND NOT   D001340.A	// R_3rd BD Z WARNING
AND NOT   D001340.C	// R_3rd BD Z SVD ERR
AND NOT   M02183	// T)R_3rd_18 Z SERVO ON
AND NOT   M00600	// EMERGENCY ALARM
OUT       D002340.1	// R_3rd BD Z SERVO ON
; L89
LOAD      M0318C	// R_3rd_18 Z Pos HOME >
OUT       D002340.4	// R_3rd BD Z HOME->
; L90
LOAD NOT  M03180	// R_3rd_18 Z Pos.1st UP >
AND NOT   M01685	// R_3rd BD Z INITIAL ->
NOT
DMOV      D004800 D002352	// R_3rd BD Z ¡Æ¢®¨ùO
DMOV      D004820 D002354	// R_3rd BD Z ¡Æ¡§¨ùO
DMOV      D004840 D002342	// R_3rd BD Z ¢¬nC¡ÍA¡×A¢®
DMOV      D004860 D002344	// R_3rd BD Z ¢¬nC¡Í¨ùO¥ì¥ì
AND       M01685	// R_3rd BD Z INITIAL ->
DMOV      1000 D002344	// R_3rd BD Z ¢¬nC¡Í¨ùO¥ì¥ì
; L95
LOAD      M03181	// R_3rd_18 Z Pos.2nd CENTER >
DMOV      D004802 D002352	// R_3rd BD Z ¡Æ¢®¨ùO
DMOV      D004822 D002354	// R_3rd BD Z ¡Æ¡§¨ùO
DMOV      D004842 D002342	// R_3rd BD Z ¢¬nC¡ÍA¡×A¢®
DMOV      D004862 D002344	// R_3rd BD Z ¢¬nC¡Í¨ùO¥ì¥ì
; L99
LOAD      M03182	// R_3rd_18 Z Pos.3rd BEND.1st >
AND NOT   M1902F	// DRY RUN
DMOV      D004804 D002352	// R_3rd BD Z ¡Æ¢®¨ùO
DMOV      D004824 D002354	// R_3rd BD Z ¡Æ¡§¨ùO
DMOV      D004844 D002342	// R_3rd BD Z BENDING POS / R_3rd BD Z ¢¬nC¡ÍA¡×A¢®
DMOV      D004864 D002344	// R_3rd BD Z ¢¬nC¡Í¨ùO¥ì¥ì

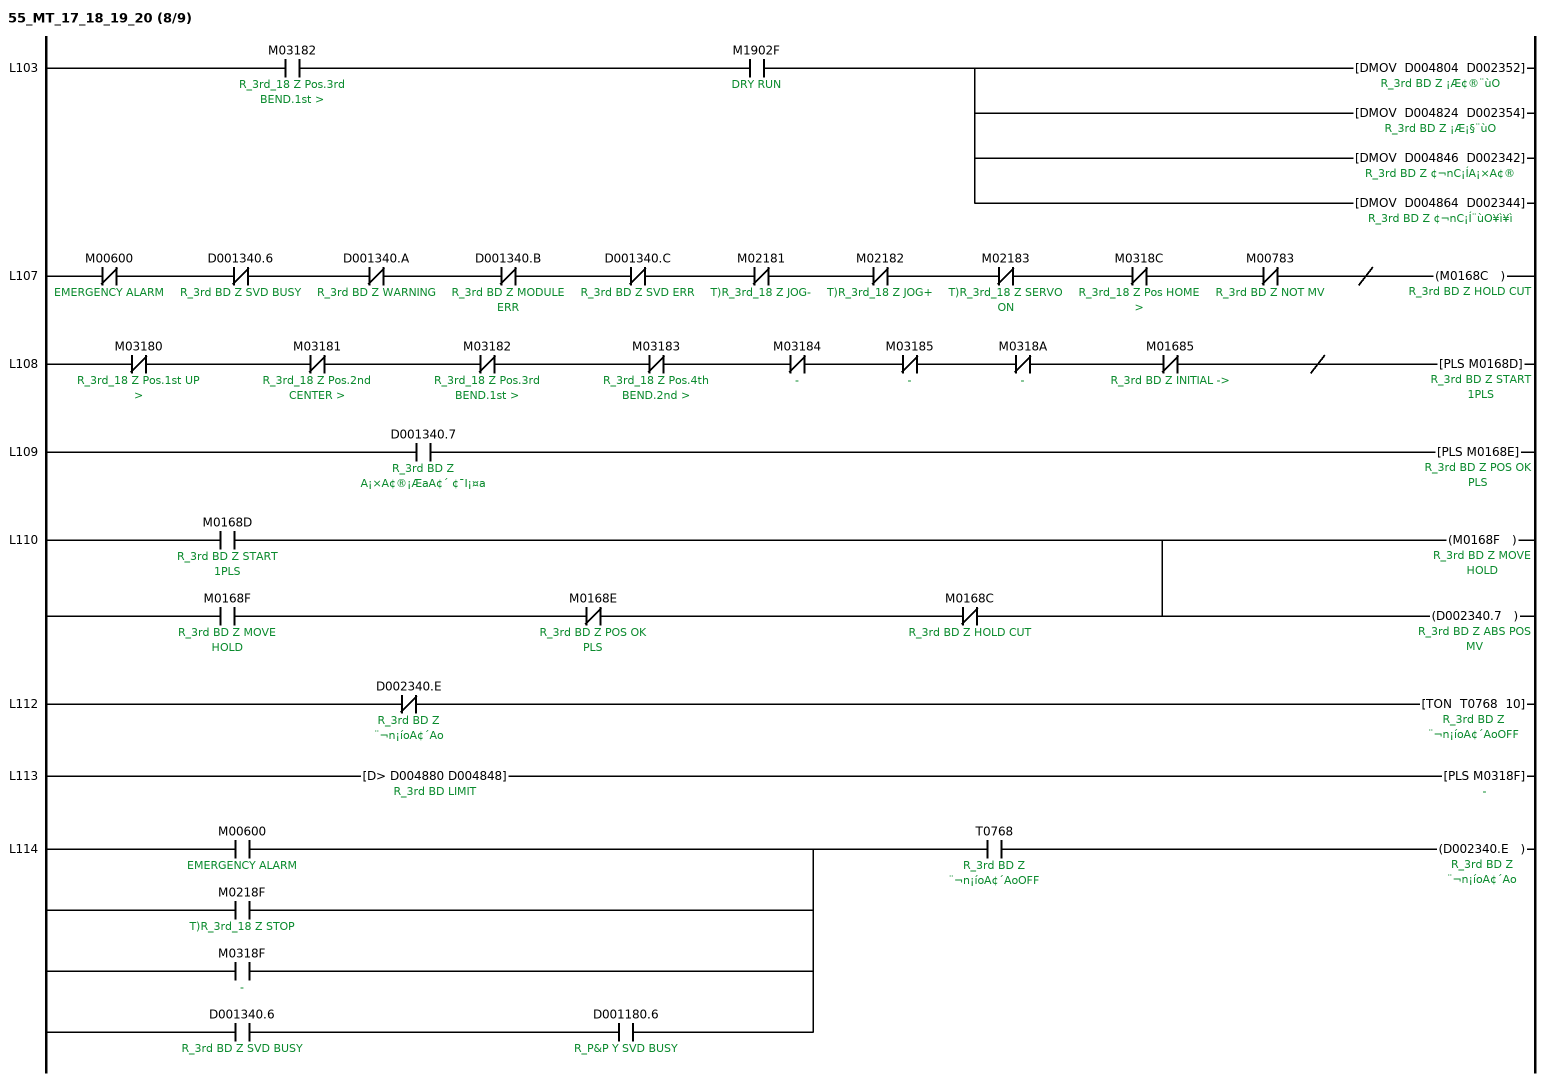
; L103
LOAD      M03182	// R_3rd_18 Z Pos.3rd BEND.1st >
AND       M1902F	// DRY RUN
DMOV      D004804 D002352	// R_3rd BD Z ¡Æ¢®¨ùO
DMOV      D004824 D002354	// R_3rd BD Z ¡Æ¡§¨ùO
DMOV      D004846 D002342	// R_3rd BD Z ¢¬nC¡ÍA¡×A¢®
DMOV      D004864 D002344	// R_3rd BD Z ¢¬nC¡Í¨ùO¥ì¥ì
; L107
LOAD NOT  M00600	// EMERGENCY ALARM
AND NOT   D001340.6	// R_3rd BD Z SVD BUSY
AND NOT   D001340.A	// R_3rd BD Z WARNING
AND NOT   D001340.B	// R_3rd BD Z MODULE ERR
AND NOT   D001340.C	// R_3rd BD Z SVD ERR
AND NOT   M02181	// T)R_3rd_18 Z JOG-
AND NOT   M02182	// T)R_3rd_18 Z JOG+
AND NOT   M02183	// T)R_3rd_18 Z SERVO ON
AND NOT   M0318C	// R_3rd_18 Z Pos HOME >
AND NOT   M00783	// R_3rd BD Z NOT MV
NOT
OUT       M0168C	// R_3rd BD Z HOLD CUT
; L108
LOAD NOT  M03180	// R_3rd_18 Z Pos.1st UP >
AND NOT   M03181	// R_3rd_18 Z Pos.2nd CENTER >
AND NOT   M03182	// R_3rd_18 Z Pos.3rd BEND.1st >
AND NOT   M03183	// R_3rd_18 Z Pos.4th BEND.2nd >
AND NOT   M03184	// -
AND NOT   M03185	// -
AND NOT   M0318A	// -
AND NOT   M01685	// R_3rd BD Z INITIAL ->
NOT
OUTP      M0168D	// R_3rd BD Z START 1PLS
; L109
LOAD      D001340.7	// R_3rd BD Z A¡×A¢®¡ÆaA¢´ ¢¯I¡¤a
OUTP      M0168E	// R_3rd BD Z POS OK PLS
; L110
LOAD      M0168D	// R_3rd BD Z START 1PLS
LOAD      M0168F	// R_3rd BD Z MOVE HOLD
AND NOT   M0168E	// R_3rd BD Z POS OK PLS
AND NOT   M0168C	// R_3rd BD Z HOLD CUT
OR LOAD
OUT       M0168F	// R_3rd BD Z MOVE HOLD
OUT       D002340.7	// R_3rd BD Z ABS POS MV
; L112
LOAD NOT  D002340.E	// R_3rd BD Z ¨¬n¡íoA¢´Ao
TON       T0768 10	// R_3rd BD Z ¨¬n¡íoA¢´AoOFF
; L113
LOADD>    D004880 D004848	// R_3rd BD LIMIT
OUTP      M0318F	// -
; L114
LOAD      M00600	// EMERGENCY ALARM
OR        M0218F	// T)R_3rd_18 Z STOP
OR        M0318F	// -
LOAD      D001340.6	// R_3rd BD Z SVD BUSY
AND       D001180.6	// R_P&P Y SVD BUSY
OR LOAD
AND       T0768	// R_3rd BD Z ¨¬n¡íoA¢´AoOFF
OUT       D002340.E	// R_3rd BD Z ¨¬n¡íoA¢´Ao

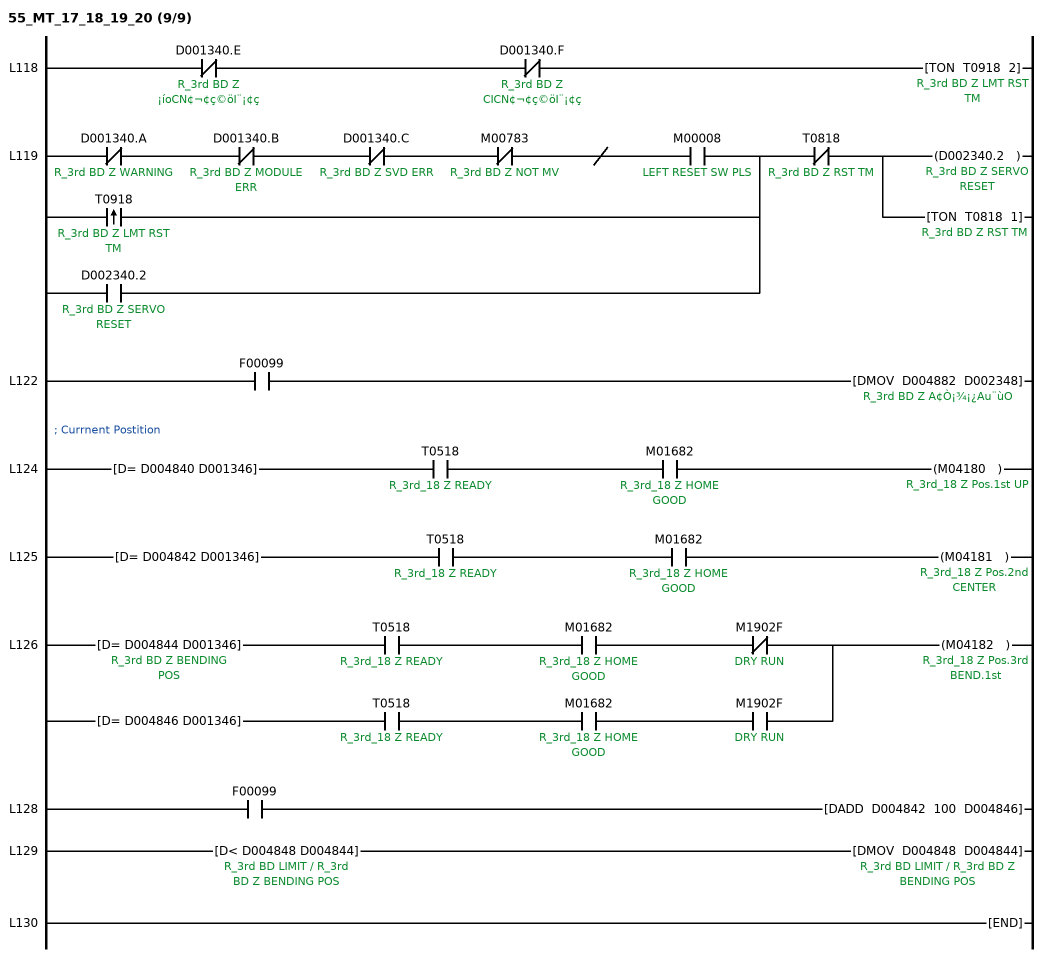
; L118
LOAD NOT  D001340.E	// R_3rd BD Z ¡íoCN¢¬¢ç©öI¨¡¢ç
AND NOT   D001340.F	// R_3rd BD Z CICN¢¬¢ç©öI¨¡¢ç
TON       T0918 2	// R_3rd BD Z LMT RST TM
; L119
LOAD NOT  D001340.A	// R_3rd BD Z WARNING
AND NOT   D001340.B	// R_3rd BD Z MODULE ERR
AND NOT   D001340.C	// R_3rd BD Z SVD ERR
AND NOT   M00783	// R_3rd BD Z NOT MV
NOT
AND       M00008	// LEFT RESET SW PLS
ORP       T0918	// R_3rd BD Z LMT RST TM
OR        D002340.2	// R_3rd BD Z SERVO RESET
AND NOT   T0818	// R_3rd BD Z RST TM
OUT       D002340.2	// R_3rd BD Z SERVO RESET
TON       T0818 1	// R_3rd BD Z RST TM
; L122
LOAD      F00099
DMOV      D004882 D002348	// R_3rd BD Z A¢Ò¡¾¡¿Au¨ùO
// Currnent Postition
; L124
LOADD=    D004840 D001346
AND       T0518	// R_3rd_18 Z READY
AND       M01682	// R_3rd_18 Z HOME GOOD
OUT       M04180	// R_3rd_18 Z Pos.1st UP
; L125
LOADD=    D004842 D001346
AND       T0518	// R_3rd_18 Z READY
AND       M01682	// R_3rd_18 Z HOME GOOD
OUT       M04181	// R_3rd_18 Z Pos.2nd CENTER
; L126
LOADD=    D004844 D001346	// R_3rd BD Z BENDING POS
AND       T0518	// R_3rd_18 Z READY
AND       M01682	// R_3rd_18 Z HOME GOOD
AND NOT   M1902F	// DRY RUN
LOADD=    D004846 D001346
AND       T0518	// R_3rd_18 Z READY
AND       M01682	// R_3rd_18 Z HOME GOOD
AND       M1902F	// DRY RUN
OR LOAD
OUT       M04182	// R_3rd_18 Z Pos.3rd BEND.1st
; L128
LOAD      F00099
DADD      D004842 100 D004846
; L129
LOADD<    D004848 D004844	// R_3rd BD LIMIT / R_3rd BD Z BENDING POS
DMOV      D004848 D004844	// R_3rd BD LIMIT / R_3rd BD Z BENDING POS
; L130
END

PROGRAM 81_OUTPUT (task: ¨ö¨¬A¥ì CA¡¤I¡¾¡¿¡¤¡Í)

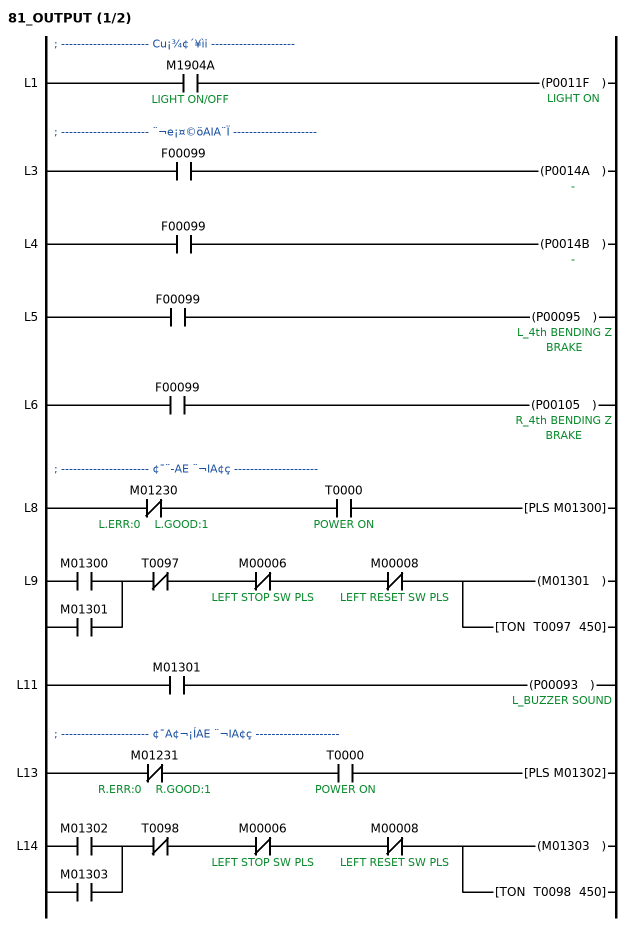
// ---------------------- Cu¡¾¢´¥ìi ---------------------
; L1
LOAD      M1904A	// LIGHT ON/OFF
OUT       P0011F	// LIGHT ON
// ---------------------- ¨¬e¡¤©öAIA¨Ï ---------------------
; L3
LOAD      F00099
OUT       P0014A	// -
; L4
LOAD      F00099
OUT       P0014B	// -
; L5
LOAD      F00099
OUT       P00095	// L_4th BENDING Z BRAKE
; L6
LOAD      F00099
OUT       P00105	// R_4th BENDING Z BRAKE
// ---------------------- ¢¯¨­AE ¨¬IA¢ç ---------------------
; L8
LOAD NOT  M01230	// L.ERR:0    L.GOOD:1
AND       T0000	// POWER ON
OUTP      M01300
; L9
LOAD      M01300
OR        M01301
AND NOT   T0097
AND NOT   M00006	// LEFT STOP SW PLS
AND NOT   M00008	// LEFT RESET SW PLS
OUT       M01301
TON       T0097 450
; L11
LOAD      M01301
OUT       P00093	// L_BUZZER SOUND
// ---------------------- ¢¯A¢¬¡ÍAE ¨¬IA¢ç ---------------------
; L13
LOAD NOT  M01231	// R.ERR:0    R.GOOD:1
AND       T0000	// POWER ON
OUTP      M01302
; L14
LOAD      M01302
OR        M01303
AND NOT   T0098
AND NOT   M00006	// LEFT STOP SW PLS
AND NOT   M00008	// LEFT RESET SW PLS
OUT       M01303
TON       T0098 450

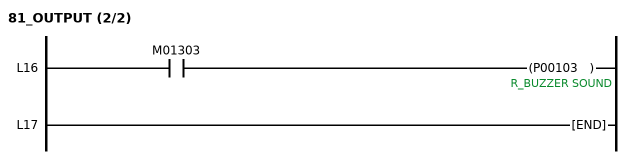
; L16
LOAD      M01303
OUT       P00103	// R_BUZZER SOUND
; L17
END

PROGRAM 82_L_MANUAL (task: ¨ö¨¬A¥ì CA¡¤I¡¾¡¿¡¤¡Í)

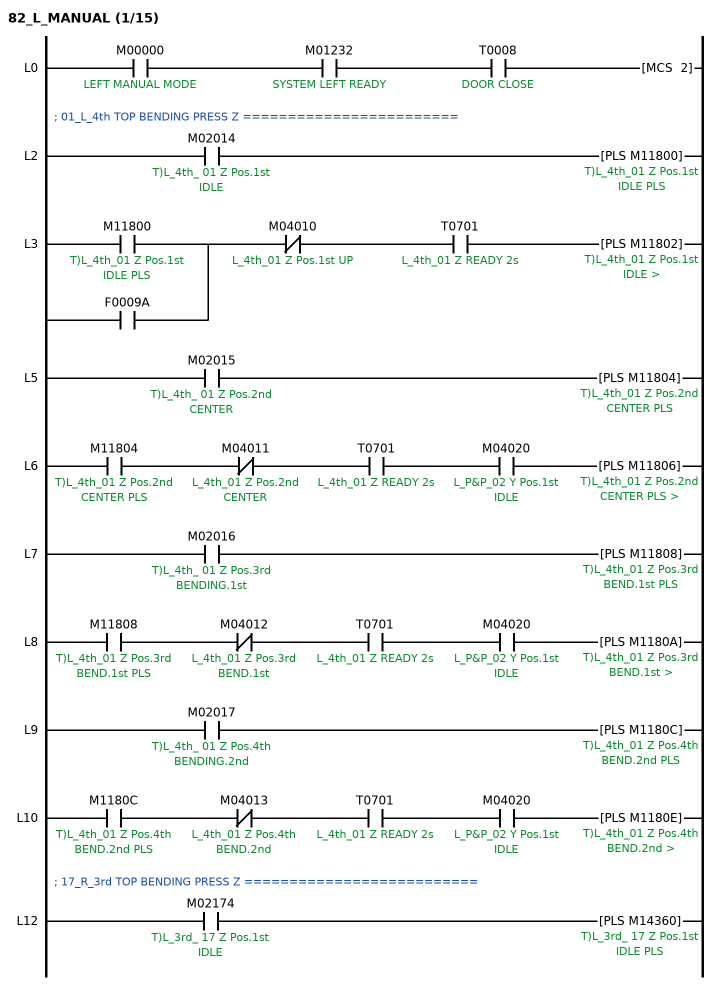
; L0
LOAD      M00000	// LEFT MANUAL MODE
AND       M01232	// SYSTEM LEFT READY
AND       T0008	// DOOR CLOSE
MCS       2
// 01_L_4th TOP BENDING PRESS Z ======================== 
; L2
LOAD      M02014	// T)L_4th_ 01 Z Pos.1st IDLE
OUTP      M11800	// T)L_4th_01 Z Pos.1st IDLE PLS
; L3
LOAD      M11800	// T)L_4th_01 Z Pos.1st IDLE PLS
OR        F0009A
AND NOT   M04010	// L_4th_01 Z Pos.1st UP
AND       T0701	// L_4th_01 Z READY 2s
OUTP      M11802	// T)L_4th_01 Z Pos.1st IDLE >
; L5
LOAD      M02015	// T)L_4th_ 01 Z Pos.2nd CENTER
OUTP      M11804	// T)L_4th_01 Z Pos.2nd CENTER PLS
; L6
LOAD      M11804	// T)L_4th_01 Z Pos.2nd CENTER PLS
AND NOT   M04011	// L_4th_01 Z Pos.2nd CENTER
AND       T0701	// L_4th_01 Z READY 2s
AND       M04020	// L_P&P_02 Y Pos.1st IDLE
OUTP      M11806	// T)L_4th_01 Z Pos.2nd CENTER PLS >
; L7
LOAD      M02016	// T)L_4th_ 01 Z Pos.3rd BENDING.1st
OUTP      M11808	// T)L_4th_01 Z Pos.3rd BEND.1st PLS
; L8
LOAD      M11808	// T)L_4th_01 Z Pos.3rd BEND.1st PLS
AND NOT   M04012	// L_4th_01 Z Pos.3rd BEND.1st
AND       T0701	// L_4th_01 Z READY 2s
AND       M04020	// L_P&P_02 Y Pos.1st IDLE
OUTP      M1180A	// T)L_4th_01 Z Pos.3rd BEND.1st >
; L9
LOAD      M02017	// T)L_4th_ 01 Z Pos.4th BENDING.2nd
OUTP      M1180C	// T)L_4th_01 Z Pos.4th BEND.2nd PLS
; L10
LOAD      M1180C	// T)L_4th_01 Z Pos.4th BEND.2nd PLS
AND NOT   M04013	// L_4th_01 Z Pos.4th BEND.2nd
AND       T0701	// L_4th_01 Z READY 2s
AND       M04020	// L_P&P_02 Y Pos.1st IDLE
OUTP      M1180E	// T)L_4th_01 Z Pos.4th BEND.2nd >
// 17_R_3rd TOP BENDING PRESS Z ==========================
; L12
LOAD      M02174	// T)L_3rd_ 17 Z Pos.1st IDLE
OUTP      M14360	// T)L_3rd_ 17 Z Pos.1st IDLE PLS

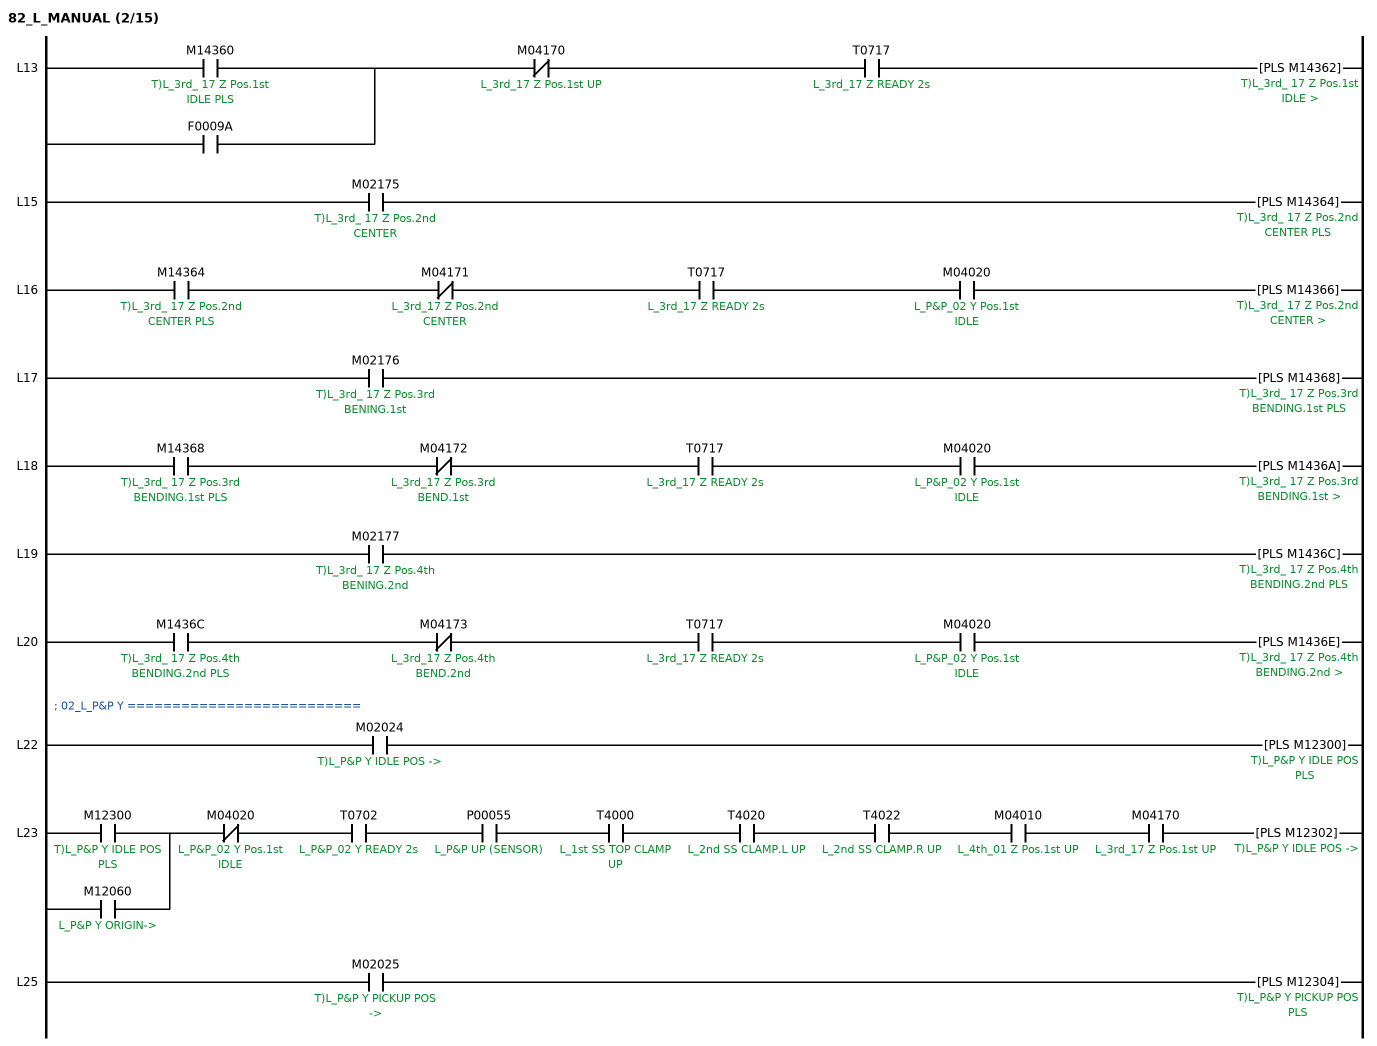
; L13
LOAD      M14360	// T)L_3rd_ 17 Z Pos.1st IDLE PLS
OR        F0009A
AND NOT   M04170	// L_3rd_17 Z Pos.1st UP
AND       T0717	// L_3rd_17 Z READY 2s
OUTP      M14362	// T)L_3rd_ 17 Z Pos.1st IDLE >
; L15
LOAD      M02175	// T)L_3rd_ 17 Z Pos.2nd CENTER
OUTP      M14364	// T)L_3rd_ 17 Z Pos.2nd CENTER PLS
; L16
LOAD      M14364	// T)L_3rd_ 17 Z Pos.2nd CENTER PLS
AND NOT   M04171	// L_3rd_17 Z Pos.2nd CENTER
AND       T0717	// L_3rd_17 Z READY 2s
AND       M04020	// L_P&P_02 Y Pos.1st IDLE
OUTP      M14366	// T)L_3rd_ 17 Z Pos.2nd CENTER >
; L17
LOAD      M02176	// T)L_3rd_ 17 Z Pos.3rd BENING.1st
OUTP      M14368	// T)L_3rd_ 17 Z Pos.3rd BENDING.1st PLS
; L18
LOAD      M14368	// T)L_3rd_ 17 Z Pos.3rd BENDING.1st PLS
AND NOT   M04172	// L_3rd_17 Z Pos.3rd BEND.1st
AND       T0717	// L_3rd_17 Z READY 2s
AND       M04020	// L_P&P_02 Y Pos.1st IDLE
OUTP      M1436A	// T)L_3rd_ 17 Z Pos.3rd BENDING.1st >
; L19
LOAD      M02177	// T)L_3rd_ 17 Z Pos.4th BENING.2nd
OUTP      M1436C	// T)L_3rd_ 17 Z Pos.4th BENDING.2nd PLS
; L20
LOAD      M1436C	// T)L_3rd_ 17 Z Pos.4th BENDING.2nd PLS
AND NOT   M04173	// L_3rd_17 Z Pos.4th BEND.2nd
AND       T0717	// L_3rd_17 Z READY 2s
AND       M04020	// L_P&P_02 Y Pos.1st IDLE
OUTP      M1436E	// T)L_3rd_ 17 Z Pos.4th BENDING.2nd >
// 02_L_P&P Y ==========================
; L22
LOAD      M02024	// T)L_P&P Y IDLE POS ->
OUTP      M12300	// T)L_P&P Y IDLE POS PLS
; L23
LOAD      M12300	// T)L_P&P Y IDLE POS PLS
OR        M12060	// L_P&P Y ORIGIN->
AND NOT   M04020	// L_P&P_02 Y Pos.1st IDLE
AND       T0702	// L_P&P_02 Y READY 2s
AND       P00055	// L_P&P UP (SENSOR)
AND       T4000	// L_1st SS TOP CLAMP    UP
AND       T4020	// L_2nd SS CLAMP.L UP
AND       T4022	// L_2nd SS CLAMP.R UP
AND       M04010	// L_4th_01 Z Pos.1st UP
AND       M04170	// L_3rd_17 Z Pos.1st UP
OUTP      M12302	// T)L_P&P Y IDLE POS ->
; L25
LOAD      M02025	// T)L_P&P Y PICKUP POS ->
OUTP      M12304	// T)L_P&P Y PICKUP POS PLS

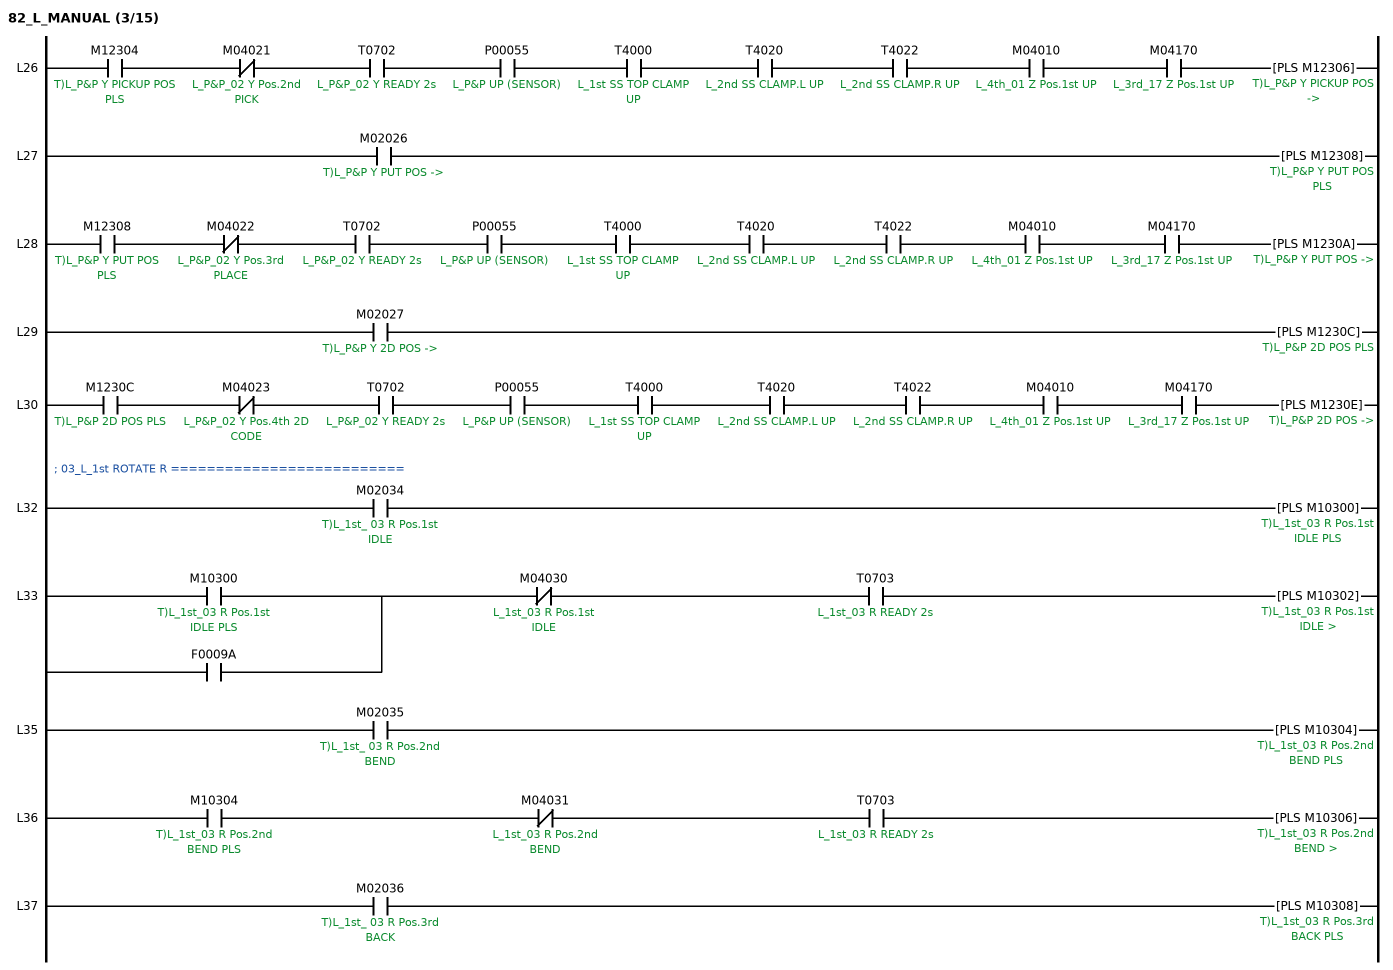
; L26
LOAD      M12304	// T)L_P&P Y PICKUP POS PLS
AND NOT   M04021	// L_P&P_02 Y Pos.2nd PICK
AND       T0702	// L_P&P_02 Y READY 2s
AND       P00055	// L_P&P UP (SENSOR)
AND       T4000	// L_1st SS TOP CLAMP    UP
AND       T4020	// L_2nd SS CLAMP.L UP
AND       T4022	// L_2nd SS CLAMP.R UP
AND       M04010	// L_4th_01 Z Pos.1st UP
AND       M04170	// L_3rd_17 Z Pos.1st UP
OUTP      M12306	// T)L_P&P Y PICKUP POS ->
; L27
LOAD      M02026	// T)L_P&P Y PUT POS ->
OUTP      M12308	// T)L_P&P Y PUT POS PLS
; L28
LOAD      M12308	// T)L_P&P Y PUT POS PLS
AND NOT   M04022	// L_P&P_02 Y Pos.3rd PLACE
AND       T0702	// L_P&P_02 Y READY 2s
AND       P00055	// L_P&P UP (SENSOR)
AND       T4000	// L_1st SS TOP CLAMP    UP
AND       T4020	// L_2nd SS CLAMP.L UP
AND       T4022	// L_2nd SS CLAMP.R UP
AND       M04010	// L_4th_01 Z Pos.1st UP
AND       M04170	// L_3rd_17 Z Pos.1st UP
OUTP      M1230A	// T)L_P&P Y PUT POS ->
; L29
LOAD      M02027	// T)L_P&P Y 2D POS ->
OUTP      M1230C	// T)L_P&P 2D POS PLS
; L30
LOAD      M1230C	// T)L_P&P 2D POS PLS
AND NOT   M04023	// L_P&P_02 Y Pos.4th 2D CODE
AND       T0702	// L_P&P_02 Y READY 2s
AND       P00055	// L_P&P UP (SENSOR)
AND       T4000	// L_1st SS TOP CLAMP    UP
AND       T4020	// L_2nd SS CLAMP.L UP
AND       T4022	// L_2nd SS CLAMP.R UP
AND       M04010	// L_4th_01 Z Pos.1st UP
AND       M04170	// L_3rd_17 Z Pos.1st UP
OUTP      M1230E	// T)L_P&P 2D POS ->
// 03_L_1st ROTATE R ==========================
; L32
LOAD      M02034	// T)L_1st_ 03 R Pos.1st IDLE
OUTP      M10300	// T)L_1st_03 R Pos.1st IDLE PLS
; L33
LOAD      M10300	// T)L_1st_03 R Pos.1st IDLE PLS
OR        F0009A
AND NOT   M04030	// L_1st_03 R Pos.1st IDLE
AND       T0703	// L_1st_03 R READY 2s
OUTP      M10302	// T)L_1st_03 R Pos.1st IDLE >
; L35
LOAD      M02035	// T)L_1st_ 03 R Pos.2nd BEND
OUTP      M10304	// T)L_1st_03 R Pos.2nd BEND PLS
; L36
LOAD      M10304	// T)L_1st_03 R Pos.2nd BEND PLS
AND NOT   M04031	// L_1st_03 R Pos.2nd BEND
AND       T0703	// L_1st_03 R READY 2s
OUTP      M10306	// T)L_1st_03 R Pos.2nd BEND >
; L37
LOAD      M02036	// T)L_1st_ 03 R Pos.3rd BACK
OUTP      M10308	// T)L_1st_03 R Pos.3rd BACK PLS

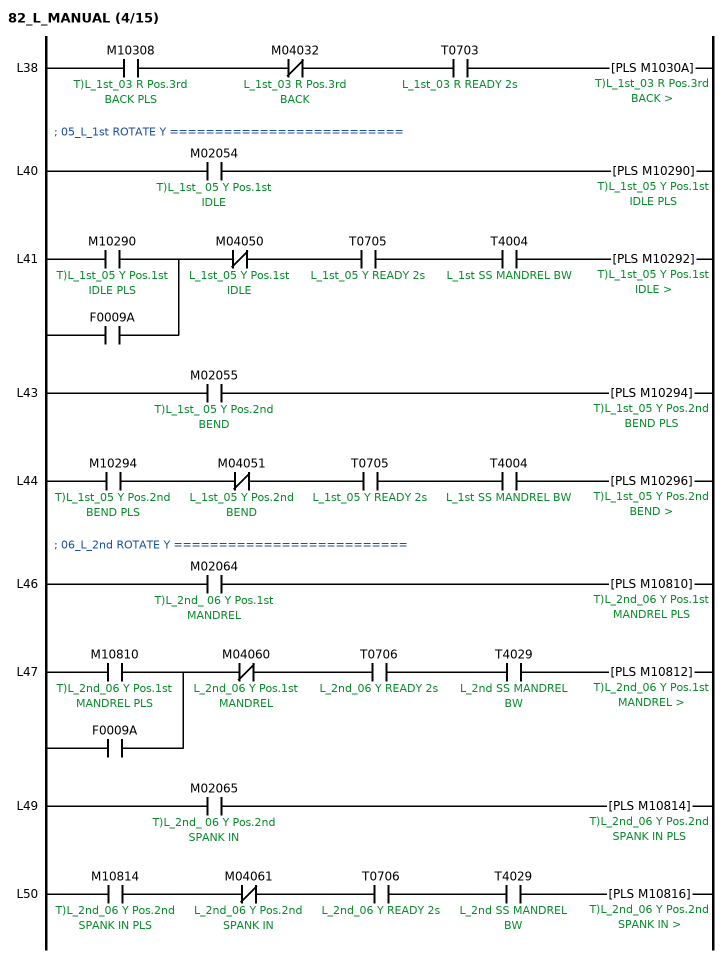
; L38
LOAD      M10308	// T)L_1st_03 R Pos.3rd BACK PLS
AND NOT   M04032	// L_1st_03 R Pos.3rd BACK
AND       T0703	// L_1st_03 R READY 2s
OUTP      M1030A	// T)L_1st_03 R Pos.3rd BACK >
// 05_L_1st ROTATE Y ==========================
; L40
LOAD      M02054	// T)L_1st_ 05 Y Pos.1st IDLE
OUTP      M10290	// T)L_1st_05 Y Pos.1st IDLE PLS
; L41
LOAD      M10290	// T)L_1st_05 Y Pos.1st IDLE PLS
OR        F0009A
AND NOT   M04050	// L_1st_05 Y Pos.1st IDLE
AND       T0705	// L_1st_05 Y READY 2s
AND       T4004	// L_1st SS MANDREL BW
OUTP      M10292	// T)L_1st_05 Y Pos.1st IDLE >
; L43
LOAD      M02055	// T)L_1st_ 05 Y Pos.2nd BEND
OUTP      M10294	// T)L_1st_05 Y Pos.2nd BEND PLS
; L44
LOAD      M10294	// T)L_1st_05 Y Pos.2nd BEND PLS
AND NOT   M04051	// L_1st_05 Y Pos.2nd BEND
AND       T0705	// L_1st_05 Y READY 2s
AND       T4004	// L_1st SS MANDREL BW
OUTP      M10296	// T)L_1st_05 Y Pos.2nd BEND >
// 06_L_2nd ROTATE Y ==========================
; L46
LOAD      M02064	// T)L_2nd_ 06 Y Pos.1st MANDREL
OUTP      M10810	// T)L_2nd_06 Y Pos.1st MANDREL PLS
; L47
LOAD      M10810	// T)L_2nd_06 Y Pos.1st MANDREL PLS
OR        F0009A
AND NOT   M04060	// L_2nd_06 Y Pos.1st MANDREL
AND       T0706	// L_2nd_06 Y READY 2s
AND       T4029	// L_2nd SS MANDREL BW
OUTP      M10812	// T)L_2nd_06 Y Pos.1st MANDREL >
; L49
LOAD      M02065	// T)L_2nd_ 06 Y Pos.2nd SPANK IN
OUTP      M10814	// T)L_2nd_06 Y Pos.2nd SPANK IN PLS
; L50
LOAD      M10814	// T)L_2nd_06 Y Pos.2nd SPANK IN PLS
AND NOT   M04061	// L_2nd_06 Y Pos.2nd SPANK IN
AND       T0706	// L_2nd_06 Y READY 2s
AND       T4029	// L_2nd SS MANDREL BW
OUTP      M10816	// T)L_2nd_06 Y Pos.2nd SPANK IN >

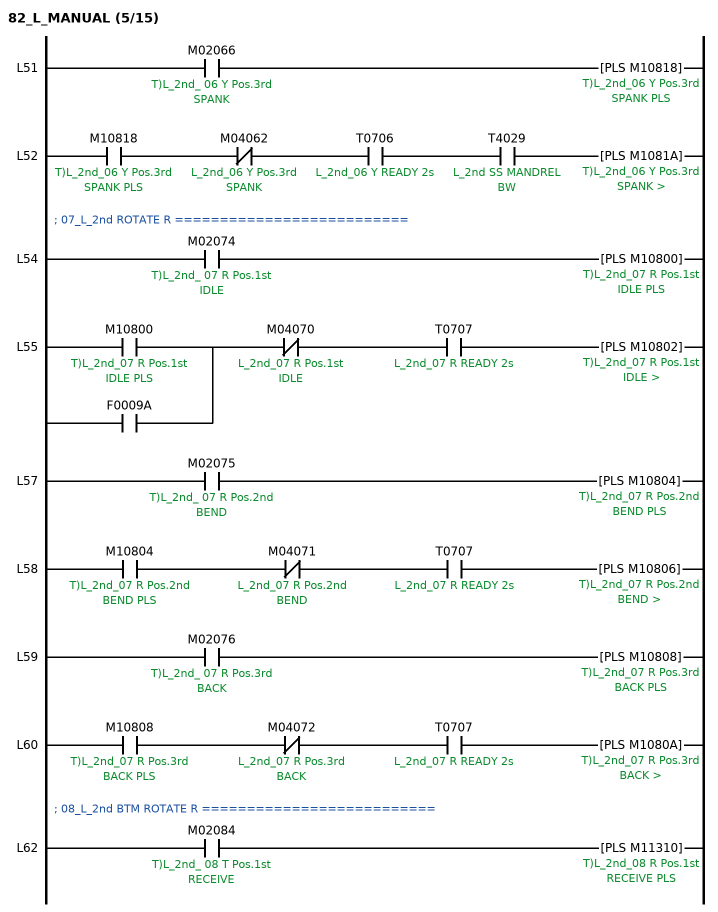
; L51
LOAD      M02066	// T)L_2nd_ 06 Y Pos.3rd SPANK
OUTP      M10818	// T)L_2nd_06 Y Pos.3rd SPANK PLS
; L52
LOAD      M10818	// T)L_2nd_06 Y Pos.3rd SPANK PLS
AND NOT   M04062	// L_2nd_06 Y Pos.3rd SPANK
AND       T0706	// L_2nd_06 Y READY 2s
AND       T4029	// L_2nd SS MANDREL BW
OUTP      M1081A	// T)L_2nd_06 Y Pos.3rd SPANK >
// 07_L_2nd ROTATE R ==========================
; L54
LOAD      M02074	// T)L_2nd_ 07 R Pos.1st IDLE
OUTP      M10800	// T)L_2nd_07 R Pos.1st IDLE PLS
; L55
LOAD      M10800	// T)L_2nd_07 R Pos.1st IDLE PLS
OR        F0009A
AND NOT   M04070	// L_2nd_07 R Pos.1st IDLE
AND       T0707	// L_2nd_07 R READY 2s
OUTP      M10802	// T)L_2nd_07 R Pos.1st IDLE >
; L57
LOAD      M02075	// T)L_2nd_ 07 R Pos.2nd BEND
OUTP      M10804	// T)L_2nd_07 R Pos.2nd BEND PLS
; L58
LOAD      M10804	// T)L_2nd_07 R Pos.2nd BEND PLS
AND NOT   M04071	// L_2nd_07 R Pos.2nd BEND
AND       T0707	// L_2nd_07 R READY 2s
OUTP      M10806	// T)L_2nd_07 R Pos.2nd BEND >
; L59
LOAD      M02076	// T)L_2nd_ 07 R Pos.3rd BACK
OUTP      M10808	// T)L_2nd_07 R Pos.3rd BACK PLS
; L60
LOAD      M10808	// T)L_2nd_07 R Pos.3rd BACK PLS
AND NOT   M04072	// L_2nd_07 R Pos.3rd BACK
AND       T0707	// L_2nd_07 R READY 2s
OUTP      M1080A	// T)L_2nd_07 R Pos.3rd BACK >
// 08_L_2nd BTM ROTATE R ==========================
; L62
LOAD      M02084	// T)L_2nd_ 08 T Pos.1st RECEIVE
OUTP      M11310	// T)L_2nd_08 R Pos.1st RECEIVE PLS

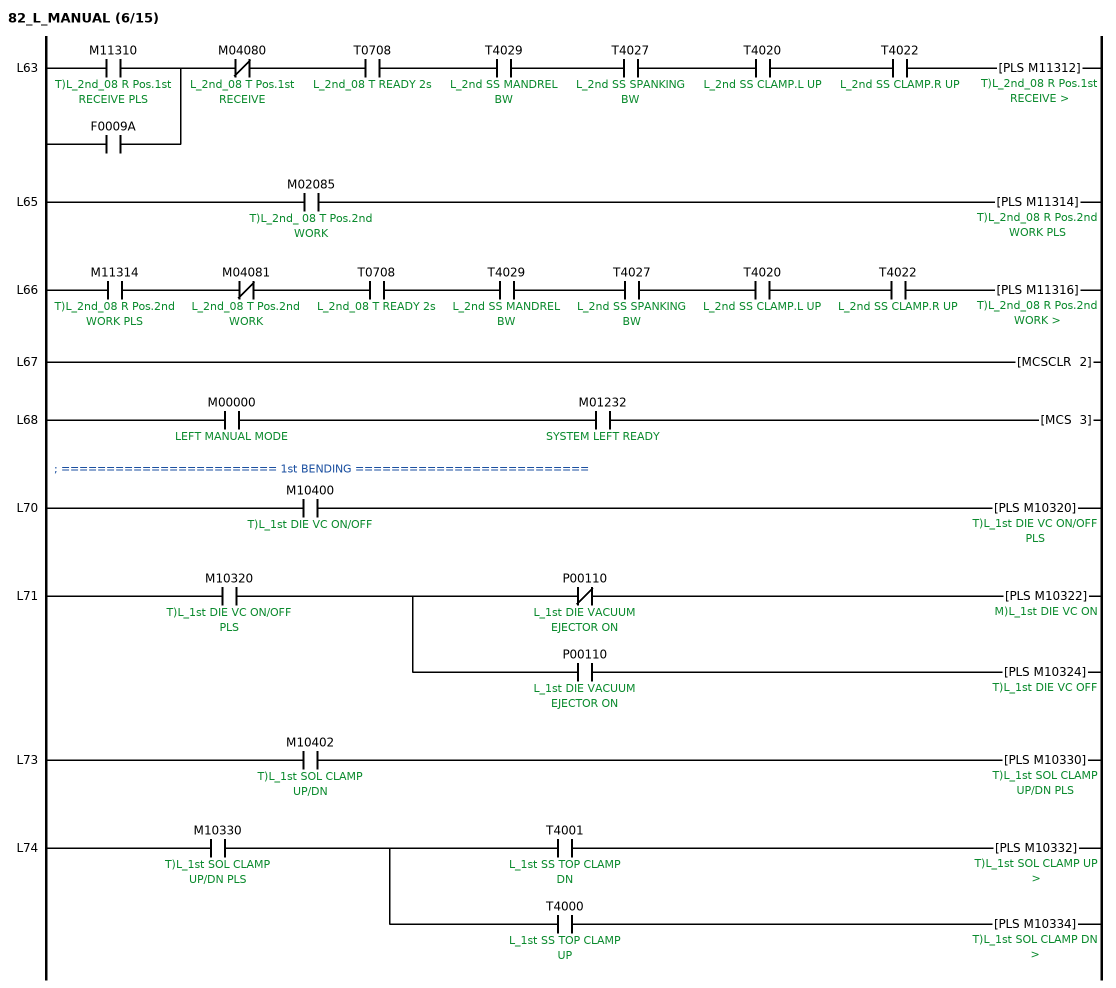
; L63
LOAD      M11310	// T)L_2nd_08 R Pos.1st RECEIVE PLS
OR        F0009A
AND NOT   M04080	// L_2nd_08 T Pos.1st RECEIVE
AND       T0708	// L_2nd_08 T READY 2s
AND       T4029	// L_2nd SS MANDREL BW
AND       T4027	// L_2nd SS SPANKING BW
AND       T4020	// L_2nd SS CLAMP.L UP
AND       T4022	// L_2nd SS CLAMP.R UP
OUTP      M11312	// T)L_2nd_08 R Pos.1st RECEIVE >
; L65
LOAD      M02085	// T)L_2nd_ 08 T Pos.2nd WORK
OUTP      M11314	// T)L_2nd_08 R Pos.2nd WORK PLS
; L66
LOAD      M11314	// T)L_2nd_08 R Pos.2nd WORK PLS
AND NOT   M04081	// L_2nd_08 T Pos.2nd WORK
AND       T0708	// L_2nd_08 T READY 2s
AND       T4029	// L_2nd SS MANDREL BW
AND       T4027	// L_2nd SS SPANKING BW
AND       T4020	// L_2nd SS CLAMP.L UP
AND       T4022	// L_2nd SS CLAMP.R UP
OUTP      M11316	// T)L_2nd_08 R Pos.2nd WORK >
; L67
MCSCLR    2
; L68
LOAD      M00000	// LEFT MANUAL MODE
AND       M01232	// SYSTEM LEFT READY
MCS       3
// ======================== 1st BENDING ==========================
; L70
LOAD      M10400	// T)L_1st DIE VC ON/OFF
OUTP      M10320	// T)L_1st DIE VC ON/OFF PLS
; L71
LOAD      M10320	// T)L_1st DIE VC ON/OFF PLS
MPUSH
AND NOT   P00110	// L_1st DIE VACUUM EJECTOR ON
OUTP      M10322	// M)L_1st DIE VC ON
MPOP
AND       P00110	// L_1st DIE VACUUM EJECTOR ON
OUTP      M10324	// T)L_1st DIE VC OFF
; L73
LOAD      M10402	// T)L_1st SOL CLAMP UP/DN
OUTP      M10330	// T)L_1st SOL CLAMP UP/DN PLS
; L74
LOAD      M10330	// T)L_1st SOL CLAMP UP/DN PLS
MPUSH
AND       T4001	// L_1st SS TOP CLAMP    DN
OUTP      M10332	// T)L_1st SOL CLAMP UP >
MPOP
AND       T4000	// L_1st SS TOP CLAMP    UP
OUTP      M10334	// T)L_1st SOL CLAMP DN >

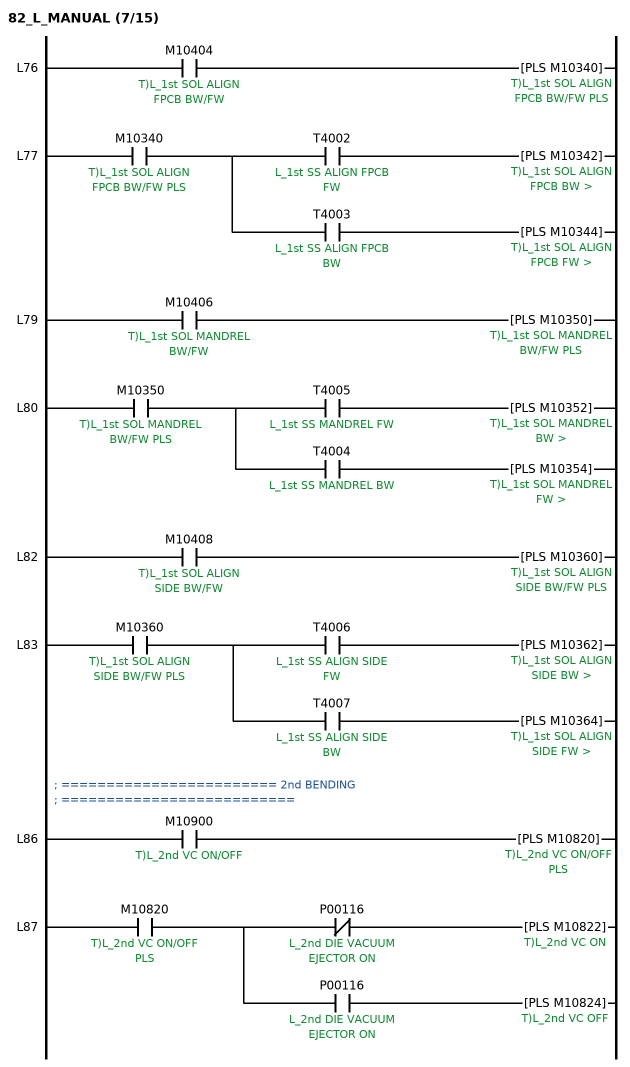
; L76
LOAD      M10404	// T)L_1st SOL ALIGN FPCB BW/FW
OUTP      M10340	// T)L_1st SOL ALIGN FPCB BW/FW PLS
; L77
LOAD      M10340	// T)L_1st SOL ALIGN FPCB BW/FW PLS
MPUSH
AND       T4002	// L_1st SS ALIGN FPCB FW
OUTP      M10342	// T)L_1st SOL ALIGN FPCB BW >
MPOP
AND       T4003	// L_1st SS ALIGN FPCB BW
OUTP      M10344	// T)L_1st SOL ALIGN FPCB FW >
; L79
LOAD      M10406	// T)L_1st SOL MANDREL BW/FW
OUTP      M10350	// T)L_1st SOL MANDREL BW/FW PLS
; L80
LOAD      M10350	// T)L_1st SOL MANDREL BW/FW PLS
MPUSH
AND       T4005	// L_1st SS MANDREL FW
OUTP      M10352	// T)L_1st SOL MANDREL BW >
MPOP
AND       T4004	// L_1st SS MANDREL BW
OUTP      M10354	// T)L_1st SOL MANDREL FW >
; L82
LOAD      M10408	// T)L_1st SOL ALIGN SIDE BW/FW
OUTP      M10360	// T)L_1st SOL ALIGN SIDE BW/FW PLS
; L83
LOAD      M10360	// T)L_1st SOL ALIGN SIDE BW/FW PLS
MPUSH
AND       T4006	// L_1st SS ALIGN SIDE FW
OUTP      M10362	// T)L_1st SOL ALIGN SIDE BW >
MPOP
AND       T4007	// L_1st SS ALIGN SIDE BW
OUTP      M10364	// T)L_1st SOL ALIGN SIDE FW >
// ======================== 2nd BENDING ==========================
; L86
LOAD      M10900	// T)L_2nd VC ON/OFF
OUTP      M10820	// T)L_2nd VC ON/OFF PLS
; L87
LOAD      M10820	// T)L_2nd VC ON/OFF PLS
MPUSH
AND NOT   P00116	// L_2nd DIE VACUUM EJECTOR ON
OUTP      M10822	// T)L_2nd VC ON
MPOP
AND       P00116	// L_2nd DIE VACUUM EJECTOR ON
OUTP      M10824	// T)L_2nd VC OFF

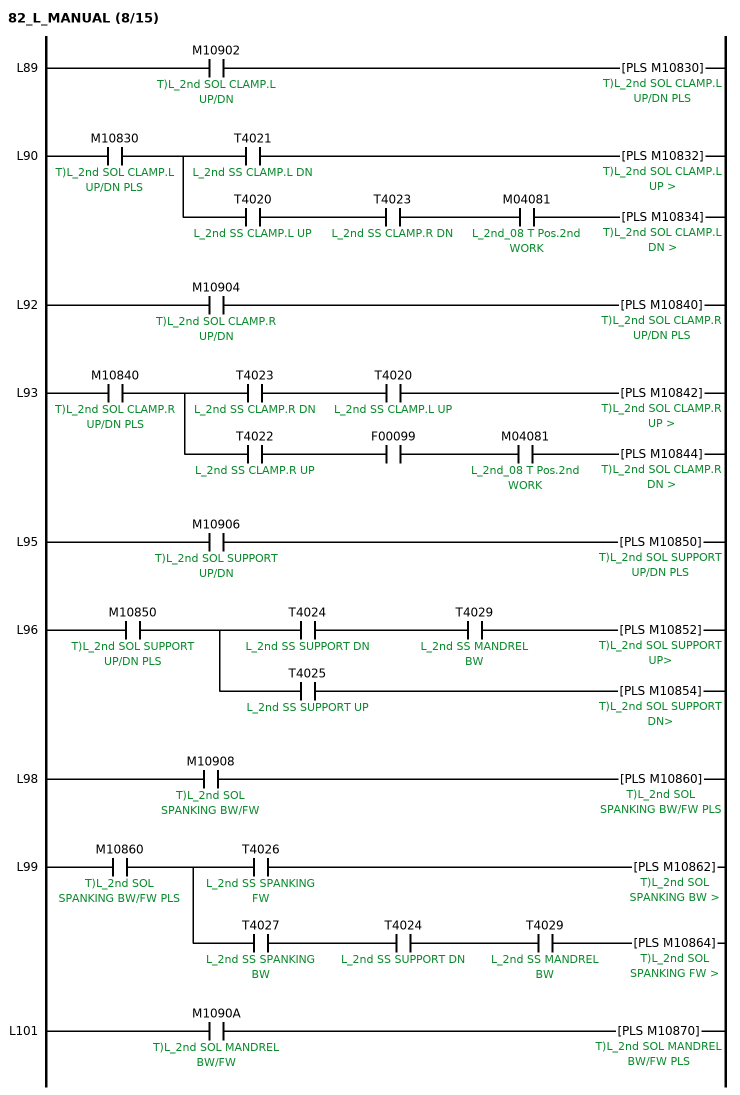
; L89
LOAD      M10902	// T)L_2nd SOL CLAMP.L UP/DN
OUTP      M10830	// T)L_2nd SOL CLAMP.L UP/DN PLS
; L90
LOAD      M10830	// T)L_2nd SOL CLAMP.L UP/DN PLS
MPUSH
AND       T4021	// L_2nd SS CLAMP.L DN
OUTP      M10832	// T)L_2nd SOL CLAMP.L UP >
MPOP
AND       T4020	// L_2nd SS CLAMP.L UP
AND       T4023	// L_2nd SS CLAMP.R DN
AND       M04081	// L_2nd_08 T Pos.2nd WORK
OUTP      M10834	// T)L_2nd SOL CLAMP.L DN >
; L92
LOAD      M10904	// T)L_2nd SOL CLAMP.R UP/DN
OUTP      M10840	// T)L_2nd SOL CLAMP.R UP/DN PLS
; L93
LOAD      M10840	// T)L_2nd SOL CLAMP.R UP/DN PLS
MPUSH
AND       T4023	// L_2nd SS CLAMP.R DN
AND       T4020	// L_2nd SS CLAMP.L UP
OUTP      M10842	// T)L_2nd SOL CLAMP.R UP >
MPOP
AND       T4022	// L_2nd SS CLAMP.R UP
AND       F00099
AND       M04081	// L_2nd_08 T Pos.2nd WORK
OUTP      M10844	// T)L_2nd SOL CLAMP.R DN >
; L95
LOAD      M10906	// T)L_2nd SOL SUPPORT UP/DN
OUTP      M10850	// T)L_2nd SOL SUPPORT UP/DN PLS
; L96
LOAD      M10850	// T)L_2nd SOL SUPPORT UP/DN PLS
MPUSH
AND       T4024	// L_2nd SS SUPPORT DN
AND       T4029	// L_2nd SS MANDREL BW
OUTP      M10852	// T)L_2nd SOL SUPPORT UP>
MPOP
AND       T4025	// L_2nd SS SUPPORT UP
OUTP      M10854	// T)L_2nd SOL SUPPORT DN>
; L98
LOAD      M10908	// T)L_2nd SOL SPANKING BW/FW
OUTP      M10860	// T)L_2nd SOL SPANKING BW/FW PLS
; L99
LOAD      M10860	// T)L_2nd SOL SPANKING BW/FW PLS
MPUSH
AND       T4026	// L_2nd SS SPANKING FW
OUTP      M10862	// T)L_2nd SOL SPANKING BW >
MPOP
AND       T4027	// L_2nd SS SPANKING BW
AND       T4024	// L_2nd SS SUPPORT DN
AND       T4029	// L_2nd SS MANDREL BW
OUTP      M10864	// T)L_2nd SOL SPANKING FW >
; L101
LOAD      M1090A	// T)L_2nd SOL MANDREL BW/FW
OUTP      M10870	// T)L_2nd SOL MANDREL BW/FW PLS

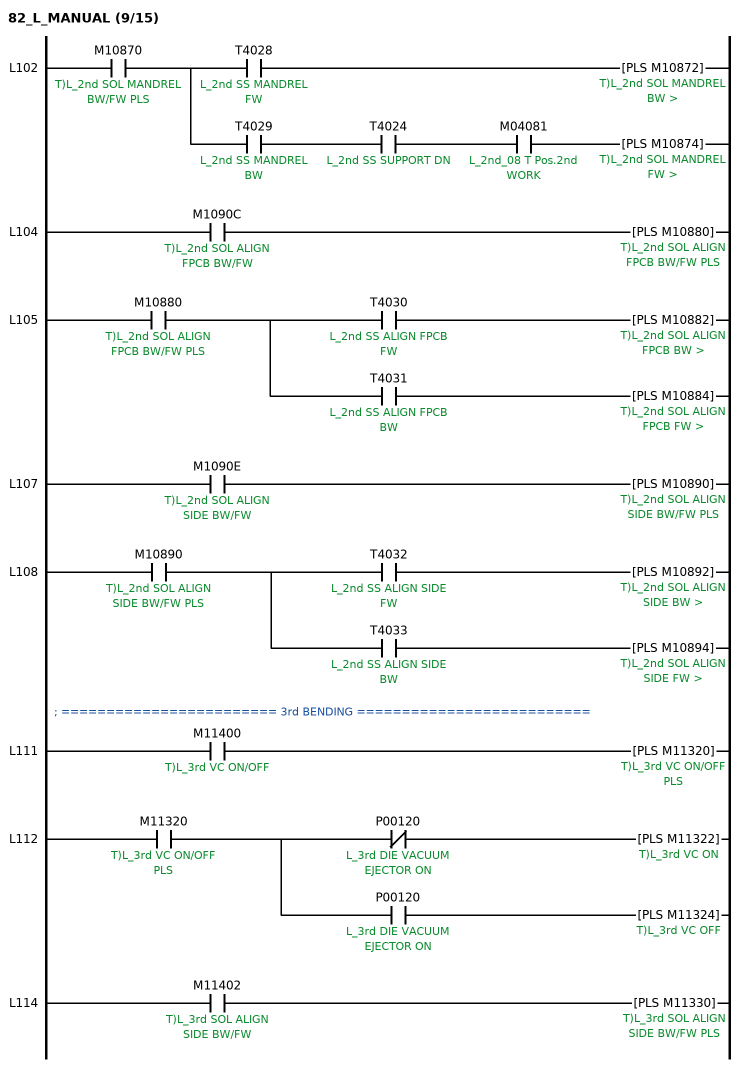
; L102
LOAD      M10870	// T)L_2nd SOL MANDREL BW/FW PLS
MPUSH
AND       T4028	// L_2nd SS MANDREL FW
OUTP      M10872	// T)L_2nd SOL MANDREL BW >
MPOP
AND       T4029	// L_2nd SS MANDREL BW
AND       T4024	// L_2nd SS SUPPORT DN
AND       M04081	// L_2nd_08 T Pos.2nd WORK
OUTP      M10874	// T)L_2nd SOL MANDREL FW >
; L104
LOAD      M1090C	// T)L_2nd SOL ALIGN FPCB BW/FW
OUTP      M10880	// T)L_2nd SOL ALIGN FPCB BW/FW PLS
; L105
LOAD      M10880	// T)L_2nd SOL ALIGN FPCB BW/FW PLS
MPUSH
AND       T4030	// L_2nd SS ALIGN FPCB FW
OUTP      M10882	// T)L_2nd SOL ALIGN FPCB BW >
MPOP
AND       T4031	// L_2nd SS ALIGN FPCB BW
OUTP      M10884	// T)L_2nd SOL ALIGN FPCB FW >
; L107
LOAD      M1090E	// T)L_2nd SOL ALIGN SIDE BW/FW
OUTP      M10890	// T)L_2nd SOL ALIGN SIDE BW/FW PLS
; L108
LOAD      M10890	// T)L_2nd SOL ALIGN SIDE BW/FW PLS
MPUSH
AND       T4032	// L_2nd SS ALIGN SIDE FW
OUTP      M10892	// T)L_2nd SOL ALIGN SIDE BW >
MPOP
AND       T4033	// L_2nd SS ALIGN SIDE BW
OUTP      M10894	// T)L_2nd SOL ALIGN SIDE FW >
// ======================== 3rd BENDING ==========================
; L111
LOAD      M11400	// T)L_3rd VC ON/OFF
OUTP      M11320	// T)L_3rd VC ON/OFF PLS
; L112
LOAD      M11320	// T)L_3rd VC ON/OFF PLS
MPUSH
AND NOT   P00120	// L_3rd DIE VACUUM EJECTOR ON
OUTP      M11322	// T)L_3rd VC ON
MPOP
AND       P00120	// L_3rd DIE VACUUM EJECTOR ON
OUTP      M11324	// T)L_3rd VC OFF
; L114
LOAD      M11402	// T)L_3rd SOL ALIGN SIDE BW/FW
OUTP      M11330	// T)L_3rd SOL ALIGN SIDE BW/FW PLS

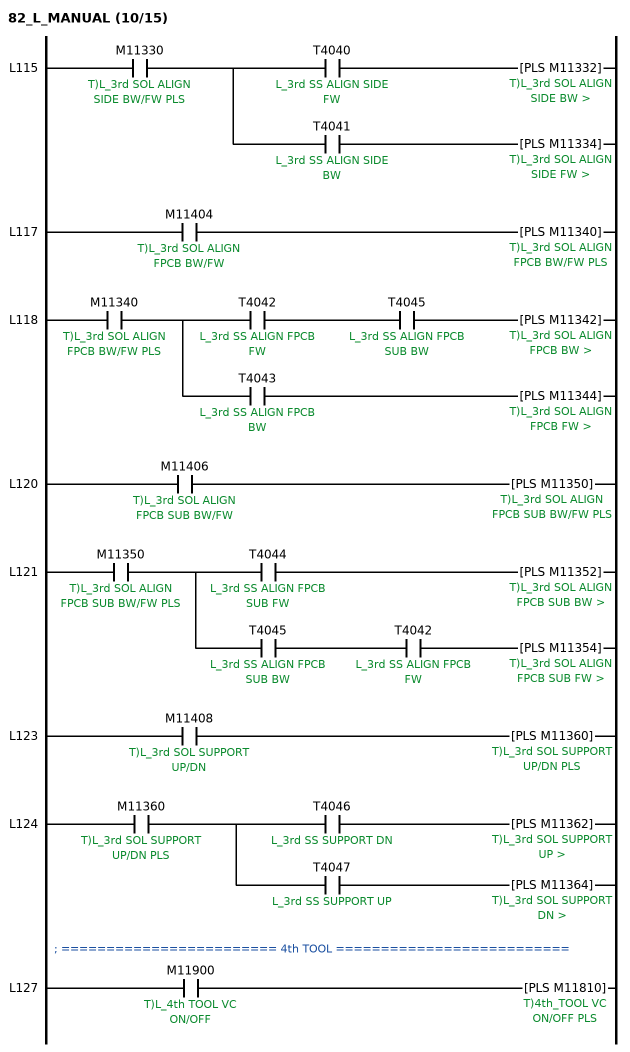
; L115
LOAD      M11330	// T)L_3rd SOL ALIGN SIDE BW/FW PLS
MPUSH
AND       T4040	// L_3rd SS ALIGN SIDE FW
OUTP      M11332	// T)L_3rd SOL ALIGN SIDE BW >
MPOP
AND       T4041	// L_3rd SS ALIGN SIDE BW
OUTP      M11334	// T)L_3rd SOL ALIGN SIDE FW >
; L117
LOAD      M11404	// T)L_3rd SOL ALIGN FPCB BW/FW
OUTP      M11340	// T)L_3rd SOL ALIGN FPCB BW/FW PLS
; L118
LOAD      M11340	// T)L_3rd SOL ALIGN FPCB BW/FW PLS
MPUSH
AND       T4042	// L_3rd SS ALIGN FPCB FW
AND       T4045	// L_3rd SS ALIGN FPCB SUB BW
OUTP      M11342	// T)L_3rd SOL ALIGN FPCB BW >
MPOP
AND       T4043	// L_3rd SS ALIGN FPCB BW
OUTP      M11344	// T)L_3rd SOL ALIGN FPCB FW >
; L120
LOAD      M11406	// T)L_3rd SOL ALIGN FPCB SUB BW/FW
OUTP      M11350	// T)L_3rd SOL ALIGN FPCB SUB BW/FW PLS
; L121
LOAD      M11350	// T)L_3rd SOL ALIGN FPCB SUB BW/FW PLS
MPUSH
AND       T4044	// L_3rd SS ALIGN FPCB SUB FW
OUTP      M11352	// T)L_3rd SOL ALIGN FPCB SUB BW >
MPOP
AND       T4045	// L_3rd SS ALIGN FPCB SUB BW
AND       T4042	// L_3rd SS ALIGN FPCB FW
OUTP      M11354	// T)L_3rd SOL ALIGN FPCB SUB FW >
; L123
LOAD      M11408	// T)L_3rd SOL SUPPORT UP/DN
OUTP      M11360	// T)L_3rd SOL SUPPORT UP/DN PLS
; L124
LOAD      M11360	// T)L_3rd SOL SUPPORT UP/DN PLS
MPUSH
AND       T4046	// L_3rd SS SUPPORT DN
OUTP      M11362	// T)L_3rd SOL SUPPORT UP >
MPOP
AND       T4047	// L_3rd SS SUPPORT UP
OUTP      M11364	// T)L_3rd SOL SUPPORT DN >
// ======================== 4th TOOL ==========================
; L127
LOAD      M11900	// T)L_4th TOOL VC ON/OFF
OUTP      M11810	// T)4th_TOOL VC ON/OFF PLS

